LIN {X 0,Y 160.848,Z 396.644,A -85,B 0,C 180,E1 -25163.822,E2 -25163.822} C_VEL
LIN {X 0,Y 156.16,Z 389.326,A -85,B 0,C 180,E1 -25166.953,E2 -25166.953} C_VEL
LIN {X 0,Y 153.521,Z 385.51,A -85,B 0,C 180,E1 -25168.906,E2 -25168.906} C_VEL
LIN {X 0,Y 150.788,Z 381.597,A -85,B 0,C 180,E1 -25171.133,E2 -25171.133} C_VEL
LIN {X 0,Y 147.963,Z 377.724,A -85,B 0,C 180,E1 -25173.701,E2 -25173.701} C_VEL
LIN {X 0,Y 145.39,Z 374.72,A -85,B 0,C 180,E1 -25176.308,E2 -25176.308} C_VEL
LIN {X 0,Y 144.413,Z 372.921,A -85,B 0,C 180,E1 -25177.489,E2 -25177.489} C_VEL
LIN {X 0,Y 141.833,Z 370.706,A -85,B 0,C 180,E1 -25180.648,E2 -25180.648} C_VEL
LIN {X 0,Y 140.04,Z 367.443,A -85,B 0,C 180,E1 -25183.603,E2 -25183.603} C_VEL
LIN {X 0,Y 137.104,Z 365.186,A -85,B 0,C 180,E1 -25189.641,E2 -25189.641} C_VEL
LIN {X 0,Y 135.74,Z 362.249,A -85,B 0,C 180,E1 -25196.661,E2 -25196.661} C_VEL
LIN {X 0,Y 135.712,Z 361.677,A -85,B 0,C 180,E1 -25200,E2 -25200} C_VEL
LIN {X 0,Y 135.941,Z 362.758,A -85,B 0,C 180,E1 -25203.334,E2 -25203.334} C_VEL
LIN {X 0,Y 139.224,Z 367.011,A -85,B 0,C 180,E1 -25213.13,E2 -25213.13} C_VEL
LIN {X 0,Y 140.214,Z 367.722,A -85,B 0,C 180,E1 -25214.792,E2 -25214.792} C_VEL
LIN {X 0,Y 142.884,Z 372.468,A -85,B 0,C 180,E1 -25218.925,E2 -25218.925} C_VEL
LIN {X 0,Y 145.937,Z 377.229,A -85,B 0,C 180,E1 -25222.593,E2 -25222.593} C_VEL
LIN {X 0,Y 149.95,Z 384.374,A -85,B 0,C 180,E1 -25226.627,E2 -25226.627} C_VEL
LIN {X 0,Y 153.462,Z 391.115,A -85,B 0,C 180,E1 -25229.653,E2 -25229.653} C_VEL
LIN {X 0,Y 156.442,Z 397.18,A -85,B 0,C 180,E1 -25231.956,E2 -25231.956} C_VEL
LIN {X 0,Y 160.501,Z 406.172,A -85,B 0,C 180,E1 -25234.811,E2 -25234.811} C_VEL
LIN {X 0,Y 165.104,Z 417.859,A -85,B 0,C 180,E1 -25237.775,E2 -25237.775} C_VEL
LIN {X 0,Y 166.456,Z 421.823,A -85,B 0,C 180,E1 -25238.615,E2 -25238.615} C_VEL
LIN {X 0,Y 167.491,Z 450.285,A -85,B 0,C 180,E1 -25240.867,E2 -25240.867} C_VEL
LIN {X 0,Y 167.692,Z 465.573,A -85,B 0,C 180,E1 -25241.895,E2 -25241.895} C_VEL
LIN {X 0,Y 166.271,Z 479.287,A -85,B 0,C 180,E1 -25242.555,E2 -25242.555} C_VEL
LIN {X 0,Y 163.763,Z 492.886,A -85,B 0,C 180,E1 -25243.599,E2 -25243.599} C_VEL
LIN {X 0,Y 160.927,Z 503.892,A -85,B 0,C 180,E1 -25244.793,E2 -25244.793} C_VEL
LIN {X 0,Y 156.98,Z 515.737,A -85,B 0,C 180,E1 -25246.502,E2 -25246.502} C_VEL
LIN {X 0,Y 152.24,Z 527.599,A -85,B 0,C 180,E1 -25248.866,E2 -25248.866} C_VEL
LIN {X 0,Y 147.198,Z 538.138,A -85,B 0,C 180,E1 -25251.634,E2 -25251.634} C_VEL
LIN {X 0,Y 142.725,Z 546.719,A -85,B 0,C 180,E1 -25254.649,E2 -25254.649} C_VEL
LIN {X 0,Y 138.004,Z 555.138,A -85,B 0,C 180,E1 -25258.535,E2 -25258.535} C_VEL
LIN {X 0,Y 134.719,Z 560.938,A -85,B 0,C 180,E1 -25261.998,E2 -25261.998} C_VEL
LIN {X 0,Y 131.482,Z 566.642,A -85,B 0,C 180,E1 -25266.367,E2 -25266.367} C_VEL
LIN {X 0,Y 129.313,Z 571.196,A -85,B 0,C 180,E1 -25270.969,E2 -25270.969} C_VEL
LIN {X 0,Y 128.07,Z 574.695,A -85,B 0,C 180,E1 -25275.704,E2 -25275.704} C_VEL
LIN {X 0,Y 127.782,Z 577.781,A -85,B 0,C 180,E1 -25281.89,E2 -25281.89} C_VEL
LIN {X 0,Y 128.495,Z 579.127,A -85,B 0,C 180,E1 -25286.865,E2 -25286.865} C_VEL
LIN {X 0,Y 129.168,Z 579.454,A -85,B 0,C 180,E1 -25290,E2 -25290} C_VEL
LIN {X 0,Y 128.502,Z 579.112,A -85,B 0,C 180,E1 -25293.135,E2 -25293.135} C_VEL
LIN {X 0,Y 127.734,Z 577.185,A -85,B 0,C 180,E1 -25299.501,E2 -25299.501} C_VEL
LIN {X 0,Y 128.056,Z 574.636,A -85,B 0,C 180,E1 -25304.298,E2 -25304.298} C_VEL
LIN {X 0,Y 129.307,Z 571.111,A -85,B 0,C 180,E1 -25309.032,E2 -25309.032} C_VEL
LIN {X 0,Y 131.492,Z 566.532,A -85,B 0,C 180,E1 -25313.631,E2 -25313.631} C_VEL
LIN {X 0,Y 134.716,Z 560.8,A -85,B 0,C 180,E1 -25318.003,E2 -25318.003} C_VEL
LIN {X 0,Y 135.726,Z 559.01,A -85,B 0,C 180,E1 -25319.152,E2 -25319.152} C_VEL
LIN {X 0,Y 136.916,Z 555.737,A -85,B 0,C 180,E1 -25321.158,E2 -25321.158} C_VEL
LIN {X 0,Y 137.589,Z 549.959,A -85,B 0,C 180,E1 -25324.523,E2 -25324.523} C_VEL
LIN {X 0,Y 138.599,Z 543.677,A -85,B 0,C 180,E1 -25327.671,E2 -25327.671} C_VEL
LIN {X 0,Y 140.244,Z 539.563,A -85,B 0,C 180,E1 -25329.273,E2 -25329.273} C_VEL
LIN {X 0,Y 145.333,Z 529.702,A -85,B 0,C 180,E1 -25332.141,E2 -25332.141} C_VEL
LIN {X 0,Y 149.725,Z 520.009,A -85,B 0,C 180,E1 -25334.284,E2 -25334.284} C_VEL
LIN {X 0,Y 153.63,Z 509.578,A -85,B 0,C 180,E1 -25336.095,E2 -25336.095} C_VEL
LIN {X 0,Y 157.496,Z 497.125,A -85,B 0,C 180,E1 -25337.651,E2 -25337.651} C_VEL
LIN {X 0,Y 160.342,Z 484.282,A -85,B 0,C 180,E1 -25338.836,E2 -25338.836} C_VEL
LIN {X 0,Y 162.321,Z 470.908,A -85,B 0,C 180,E1 -25339.636,E2 -25339.636} C_VEL
LIN {X 0,Y 162.803,Z 463.571,A -85,B 0,C 180,E1 -25339.985,E2 -25339.985} C_VEL
LIN {X 0,Y 162.131,Z 433.785,A -85,B 0,C 180,E1 -25342.28,E2 -25342.28} C_VEL
LIN {X 0,Y 161.697,Z 423.97,A -85,B 0,C 180,E1 -25343.163,E2 -25343.163} C_VEL
LIN {X 0,Y 157.863,Z 413.397,A -85,B 0,C 180,E1 -25345.802,E2 -25345.802} C_VEL
LIN {X 0,Y 154.013,Z 404.075,A -85,B 0,C 180,E1 -25348.674,E2 -25348.674} C_VEL
LIN {X 0,Y 151.004,Z 397.589,A -85,B 0,C 180,E1 -25351.127,E2 -25351.127} C_VEL
LIN {X 0,Y 148.579,Z 392.638,A -85,B 0,C 180,E1 -25353.297,E2 -25353.297} C_VEL
LIN {X 0,Y 146.169,Z 387.847,A -85,B 0,C 180,E1 -25355.689,E2 -25355.689} C_VEL
LIN {X 0,Y 142.972,Z 381.909,A -85,B 0,C 180,E1 -25359.327,E2 -25359.327} C_VEL
LIN {X 0,Y 139.556,Z 376.178,A -85,B 0,C 180,E1 -25364.155,E2 -25364.155} C_VEL
LIN {X 0,Y 138.499,Z 374.182,A -85,B 0,C 180,E1 -25366.053,E2 -25366.053} C_VEL
LIN {X 0,Y 135.372,Z 370.964,A -85,B 0,C 180,E1 -25373.479,E2 -25373.479} C_VEL
LIN {X 0,Y 134.671,Z 368.946,A -85,B 0,C 180,E1 -25377.757,E2 -25377.757} C_VEL
LIN {X 0,Y 134.53,Z 368.503,A -85,B 0,C 180,E1 -25380,E2 -25380} C_VEL
LIN {X 0,Y 134.722,Z 369.26,A -85,B 0,C 180,E1 -25384.863,E2 -25384.863} C_VEL
LIN {X 0,Y 137.525,Z 373.69,A -85,B 0,C 180,E1 -25394.237,E2 -25394.237} C_VEL
LIN {X 0,Y 138.784,Z 374.55,A -85,B 0,C 180,E1 -25396.455,E2 -25396.455} C_VEL
LIN {X 0,Y 140.616,Z 377.811,A -85,B 0,C 180,E1 -25399.48,E2 -25399.48} C_VEL
LIN {X 0,Y 142.797,Z 379.938,A -85,B 0,C 180,E1 -25402.232,E2 -25402.232} C_VEL
LIN {X 0,Y 145.118,Z 383.369,A -85,B 0,C 180,E1 -25404.893,E2 -25404.893} C_VEL
LIN {X 0,Y 146.391,Z 384.854,A -85,B 0,C 180,E1 -25406.162,E2 -25406.162} C_VEL
LIN {X 0,Y 149.998,Z 390.076,A -85,B 0,C 180,E1 -25409.47,E2 -25409.47} C_VEL
LIN {X 0,Y 152.651,Z 394,A -85,B 0,C 180,E1 -25411.612,E2 -25411.612} C_VEL
LIN {X 0,Y 157.355,Z 401.577,A -85,B 0,C 180,E1 -25415.005,E2 -25415.005} C_VEL
LIN {X 0,Y 162.803,Z 411.309,A -85,B 0,C 180,E1 -25418.448,E2 -25418.448} C_VEL
LIN {X 0,Y 166.396,Z 418.787,A -85,B 0,C 180,E1 -25420.534,E2 -25420.534} C_VEL
LIN {X 0,Y 164.916,Z 443.762,A -85,B 0,C 180,E1 -25421.725,E2 -25421.725} C_VEL
LIN {X 0,Y 163.206,Z 456.855,A -85,B 0,C 180,E1 -25422.747,E2 -25422.747} C_VEL
LIN {X 0,Y 160.816,Z 468.889,A -85,B 0,C 180,E1 -25424.107,E2 -25424.107} C_VEL
LIN {X 0,Y 157.42,Z 481.198,A -85,B 0,C 180,E1 -25425.986,E2 -25425.986} C_VEL
LIN {X 0,Y 153.617,Z 491.66,A -85,B 0,C 180,E1 -25428.004,E2 -25428.004} C_VEL
LIN {X 0,Y 149.798,Z 500.707,A -85,B 0,C 180,E1 -25430.266,E2 -25430.266} C_VEL
LIN {X 0,Y 145.875,Z 509.102,A -85,B 0,C 180,E1 -25432.971,E2 -25432.971} C_VEL
LIN {X 0,Y 141.753,Z 516.834,A -85,B 0,C 180,E1 -25436.099,E2 -25436.099} C_VEL
LIN {X 0,Y 137.219,Z 524.484,A -85,B 0,C 180,E1 -25440.127,E2 -25440.127} C_VEL
LIN {X 0,Y 132.797,Z 531.281,A -85,B 0,C 180,E1 -25444.952,E2 -25444.952} C_VEL
LIN {X 0,Y 129.504,Z 535.886,A -85,B 0,C 180,E1 -25449.345,E2 -25449.345} C_VEL
LIN {X 0,Y 126.664,Z 539.432,A -85,B 0,C 180,E1 -25453.894,E2 -25453.894} C_VEL
LIN {X 0,Y 125.228,Z 541.253,A -85,B 0,C 180,E1 -25457.028,E2 -25457.028} C_VEL
LIN {X 0,Y 124.381,Z 542.581,A -85,B 0,C 180,E1 -25460.241,E2 -25460.241} C_VEL
LIN {X 0,Y 123.277,Z 544.125,A -85,B 0,C 180,E1 -25466.732,E2 -25466.732} C_VEL
LIN {X 0,Y 123.137,Z 544.345,A -85,B 0,C 180,E1 -25470,E2 -25470} C_VEL
LIN {X 0,Y 123.276,Z 544.154,A -85,B 0,C 180,E1 -25473.268,E2 -25473.268} C_VEL
LIN {X 0,Y 124.373,Z 542.648,A -85,B 0,C 180,E1 -25479.76,E2 -25479.76} C_VEL
LIN {X 0,Y 125.21,Z 541.351,A -85,B 0,C 180,E1 -25482.974,E2 -25482.974} C_VEL
LIN {X 0,Y 127.632,Z 538.503,A -85,B 0,C 180,E1 -25487.629,E2 -25487.629} C_VEL
LIN {X 0,Y 130.589,Z 534.667,A -85,B 0,C 180,E1 -25492.131,E2 -25492.131} C_VEL
LIN {X 0,Y 134.038,Z 529.576,A -85,B 0,C 180,E1 -25496.633,E2 -25496.633} C_VEL
LIN {X 0,Y 138.751,Z 522.322,A -85,B 0,C 180,E1 -25501.277,E2 -25501.277} C_VEL
LIN {X 0,Y 143.406,Z 514.284,A -85,B 0,C 180,E1 -25505.158,E2 -25505.158} C_VEL
LIN {X 0,Y 147.564,Z 506.049,A -85,B 0,C 180,E1 -25508.253,E2 -25508.253} C_VEL
LIN {X 0,Y 151.583,Z 496.997,A -85,B 0,C 180,E1 -25510.911,E2 -25510.911} C_VEL
LIN {X 0,Y 155.836,Z 486.44,A -85,B 0,C 180,E1 -25513.208,E2 -25513.208} C_VEL
LIN {X 0,Y 159.464,Z 474.891,A -85,B 0,C 180,E1 -25515.203,E2 -25515.203} C_VEL
LIN {X 0,Y 162.311,Z 463.568,A -85,B 0,C 180,E1 -25516.648,E2 -25516.648} C_VEL
LIN {X 0,Y 164.339,Z 450.783,A -85,B 0,C 180,E1 -25517.921,E2 -25517.921} C_VEL
LIN {X 0,Y 165.583,Z 437.335,A -85,B 0,C 180,E1 -25518.794,E2 -25518.794} C_VEL
LIN {X 0,Y 166.549,Z 418.84,A -85,B 0,C 180,E1 -25519.632,E2 -25519.632} C_VEL
LIN {X 0,Y 161.33,Z 408.377,A -85,B 0,C 180,E1 -25522.708,E2 -25522.708} C_VEL
LIN {X 0,Y 156.008,Z 399.158,A -85,B 0,C 180,E1 -25526.215,E2 -25526.215} C_VEL
LIN {X 0,Y 151.502,Z 392.096,A -85,B 0,C 180,E1 -25529.62,E2 -25529.62} C_VEL
LIN {X 0,Y 148.293,Z 387.477,A -85,B 0,C 180,E1 -25532.383,E2 -25532.383} C_VEL
LIN {X 0,Y 145.945,Z 384.127,A -85,B 0,C 180,E1 -25534.67,E2 -25534.67} C_VEL
LIN {X 0,Y 143.441,Z 380.953,A -85,B 0,C 180,E1 -25537.399,E2 -25537.399} C_VEL
LIN {X 0,Y 142.436,Z 379.406,A -85,B 0,C 180,E1 -25538.66,E2 -25538.66} C_VEL
LIN {X 0,Y 139.927,Z 376.762,A -85,B 0,C 180,E1 -25542.083,E2 -25542.083} C_VEL
LIN {X 0,Y 138.767,Z 374.319,A -85,B 0,C 180,E1 -25544.209,E2 -25544.209} C_VEL
LIN {X 0,Y 135.95,Z 371.966,A -85,B 0,C 180,E1 -25550.468,E2 -25550.468} C_VEL
LIN {X 0,Y 134.849,Z 369.244,A -85,B 0,C 180,E1 -25557.012,E2 -25557.012} C_VEL
LIN {X 0,Y 134.844,Z 368.749,A -85,B 0,C 180,E1 -25560,E2 -25560} C_VEL
LIN {X 0,Y 135.018,Z 369.778,A -85,B 0,C 180,E1 -25562.984,E2 -25562.984} C_VEL
LIN {X 0,Y 138.177,Z 373.995,A -85,B 0,C 180,E1 -25572.857,E2 -25572.857} C_VEL
LIN {X 0,Y 138.967,Z 374.761,A -85,B 0,C 180,E1 -25574.273,E2 -25574.273} C_VEL
LIN {X 0,Y 143.58,Z 382.67,A -85,B 0,C 180,E1 -25581.054,E2 -25581.054} C_VEL
LIN {X 0,Y 147.51,Z 390.237,A -85,B 0,C 180,E1 -25585.391,E2 -25585.391} C_VEL
LIN {X 0,Y 150.696,Z 396.745,A -85,B 0,C 180,E1 -25588.367,E2 -25588.367} C_VEL
LIN {X 0,Y 153.679,Z 403.119,A -85,B 0,C 180,E1 -25590.847,E2 -25590.847} C_VEL
LIN {X 0,Y 157.606,Z 412.501,A -85,B 0,C 180,E1 -25593.821,E2 -25593.821} C_VEL
LIN {X 0,Y 161.436,Z 422.806,A -85,B 0,C 180,E1 -25596.478,E2 -25596.478} C_VEL
LIN {X 0,Y 162.044,Z 424.806,A -85,B 0,C 180,E1 -25596.9,E2 -25596.9} C_VEL
LIN {X 0,Y 162.863,Z 454.654,A -85,B 0,C 180,E1 -25599.307,E2 -25599.307} C_VEL
LIN {X 0,Y 162.867,Z 466.599,A -85,B 0,C 180,E1 -25600.108,E2 -25600.108} C_VEL
LIN {X 0,Y 161.199,Z 480.534,A -85,B 0,C 180,E1 -25600.842,E2 -25600.842} C_VEL
LIN {X 0,Y 158.648,Z 493.207,A -85,B 0,C 180,E1 -25601.861,E2 -25601.861} C_VEL
LIN {X 0,Y 155.421,Z 504.815,A -85,B 0,C 180,E1 -25603.185,E2 -25603.185} C_VEL
LIN {X 0,Y 151.325,Z 516.187,A -85,B 0,C 180,E1 -25604.908,E2 -25604.908} C_VEL
LIN {X 0,Y 146.97,Z 526.615,A -85,B 0,C 180,E1 -25607.046,E2 -25607.046} C_VEL
LIN {X 0,Y 141.693,Z 537.151,A -85,B 0,C 180,E1 -25609.85,E2 -25609.85} C_VEL
LIN {X 0,Y 136.951,Z 545.726,A -85,B 0,C 180,E1 -25612.917,E2 -25612.917} C_VEL
LIN {X 0,Y 131.954,Z 554.144,A -85,B 0,C 180,E1 -25616.913,E2 -25616.913} C_VEL
LIN {X 0,Y 127.402,Z 561.729,A -85,B 0,C 180,E1 -25621.777,E2 -25621.777} C_VEL
LIN {X 0,Y 124.003,Z 567.302,A -85,B 0,C 180,E1 -25626.626,E2 -25626.626} C_VEL
LIN {X 0,Y 121.965,Z 571.498,A -85,B 0,C 180,E1 -25631.523,E2 -25631.523} C_VEL
LIN {X 0,Y 120.883,Z 574.668,A -85,B 0,C 180,E1 -25636.553,E2 -25636.553} C_VEL
LIN {X 0,Y 120.739,Z 576.9,A -85,B 0,C 180,E1 -25641.705,E2 -25641.705} C_VEL
LIN {X 0,Y 121.383,Z 578.136,A -85,B 0,C 180,E1 -25646.681,E2 -25646.681} C_VEL
LIN {X 0,Y 122.079,Z 578.468,A -85,B 0,C 180,E1 -25650,E2 -25650} C_VEL
LIN {X 0,Y 121.388,Z 578.12,A -85,B 0,C 180,E1 -25653.319,E2 -25653.319} C_VEL
LIN {X 0,Y 120.685,Z 576.189,A -85,B 0,C 180,E1 -25660.061,E2 -25660.061} C_VEL
LIN {X 0,Y 121.106,Z 573.635,A -85,B 0,C 180,E1 -25665.138,E2 -25665.138} C_VEL
LIN {X 0,Y 122.552,Z 570.113,A -85,B 0,C 180,E1 -25670.125,E2 -25670.125} C_VEL
LIN {X 0,Y 124.983,Z 565.537,A -85,B 0,C 180,E1 -25674.944,E2 -25674.944} C_VEL
LIN {X 0,Y 129.103,Z 558.739,A -85,B 0,C 180,E1 -25680.234,E2 -25680.234} C_VEL
LIN {X 0,Y 133.516,Z 551.342,A -85,B 0,C 180,E1 -25684.461,E2 -25684.461} C_VEL
LIN {X 0,Y 138.779,Z 542.234,A -85,B 0,C 180,E1 -25688.342,E2 -25688.342} C_VEL
LIN {X 0,Y 140.244,Z 539.563,A -85,B 0,C 180,E1 -25689.273,E2 -25689.273} C_VEL
LIN {X 0,Y 141.932,Z 535.289,A -85,B 0,C 180,E1 -25690.783,E2 -25690.783} C_VEL
LIN {X 0,Y 143.283,Z 527.963,A -85,B 0,C 180,E1 -25693.432,E2 -25693.432} C_VEL
LIN {X 0,Y 144.624,Z 520.254,A -85,B 0,C 180,E1 -25695.852,E2 -25695.852} C_VEL
LIN {X 0,Y 146.216,Z 515.282,A -85,B 0,C 180,E1 -25696.964,E2 -25696.964} C_VEL
LIN {X 0,Y 150.611,Z 503.291,A -85,B 0,C 180,E1 -25698.801,E2 -25698.801} C_VEL
LIN {X 0,Y 153.972,Z 491.422,A -85,B 0,C 180,E1 -25700.122,E2 -25700.122} C_VEL
LIN {X 0,Y 156.705,Z 477.922,A -85,B 0,C 180,E1 -25701.169,E2 -25701.169} C_VEL
LIN {X 0,Y 158.179,Z 465.114,A -85,B 0,C 180,E1 -25701.839,E2 -25701.839} C_VEL
LIN {X 0,Y 157.764,Z 435.791,A -85,B 0,C 180,E1 -25704.154,E2 -25704.154} C_VEL
LIN {X 0,Y 157.501,Z 427.116,A -85,B 0,C 180,E1 -25704.935,E2 -25704.935} C_VEL
LIN {X 0,Y 153.986,Z 417.044,A -85,B 0,C 180,E1 -25707.598,E2 -25707.598} C_VEL
LIN {X 0,Y 150.252,Z 407.681,A -85,B 0,C 180,E1 -25710.681,E2 -25710.681} C_VEL
LIN {X 0,Y 146.701,Z 399.622,A -85,B 0,C 180,E1 -25713.982,E2 -25713.982} C_VEL
LIN {X 0,Y 144.01,Z 393.968,A -85,B 0,C 180,E1 -25716.83,E2 -25716.83} C_VEL
LIN {X 0,Y 140.882,Z 387.867,A -85,B 0,C 180,E1 -25720.701,E2 -25720.701} C_VEL
LIN {X 0,Y 138.064,Z 382.758,A -85,B 0,C 180,E1 -25725.066,E2 -25725.066} C_VEL
LIN {X 0,Y 137.038,Z 380.911,A -85,B 0,C 180,E1 -25727.034,E2 -25727.034} C_VEL
LIN {X 0,Y 134.129,Z 377.356,A -85,B 0,C 180,E1 -25735.116,E2 -25735.116} C_VEL
LIN {X 0,Y 133.735,Z 375.85,A -85,B 0,C 180,E1 -25738.494,E2 -25738.494} C_VEL
LIN {X 0,Y 133.663,Z 375.564,A -85,B 0,C 180,E1 -25740,E2 -25740} C_VEL
LIN {X 0,Y 133.848,Z 376.404,A -85,B 0,C 180,E1 -25744.895,E2 -25744.895} C_VEL
LIN {X 0,Y 136.403,Z 380.62,A -85,B 0,C 180,E1 -25753.786,E2 -25753.786} C_VEL
LIN {X 0,Y 137.446,Z 381.457,A -85,B 0,C 180,E1 -25755.748,E2 -25755.748} C_VEL
LIN {X 0,Y 139.422,Z 384.832,A -85,B 0,C 180,E1 -25759.127,E2 -25759.127} C_VEL
LIN {X 0,Y 141.041,Z 386.461,A -85,B 0,C 180,E1 -25761.274,E2 -25761.274} C_VEL
LIN {X 0,Y 143.596,Z 390.188,A -85,B 0,C 180,E1 -25764.34,E2 -25764.34} C_VEL
LIN {X 0,Y 147.428,Z 395.805,A -85,B 0,C 180,E1 -25768.174,E2 -25768.174} C_VEL
LIN {X 0,Y 151.366,Z 401.899,A -85,B 0,C 180,E1 -25771.511,E2 -25771.511} C_VEL
LIN {X 0,Y 156.637,Z 411.198,A -85,B 0,C 180,E1 -25775.386,E2 -25775.386} C_VEL
LIN {X 0,Y 161.17,Z 420.199,A -85,B 0,C 180,E1 -25778.328,E2 -25778.328} C_VEL
LIN {X 0,Y 161.803,Z 421.629,A -85,B 0,C 180,E1 -25778.722,E2 -25778.722} C_VEL
LIN {X 0,Y 160.385,Z 444.105,A -85,B 0,C 180,E1 -25779.805,E2 -25779.805} C_VEL
LIN {X 0,Y 158.539,Z 457.708,A -85,B 0,C 180,E1 -25780.868,E2 -25780.868} C_VEL
LIN {X 0,Y 156.006,Z 469.873,A -85,B 0,C 180,E1 -25782.253,E2 -25782.253} C_VEL
LIN {X 0,Y 152.442,Z 482.184,A -85,B 0,C 180,E1 -25784.15,E2 -25784.15} C_VEL
LIN {X 0,Y 148.468,Z 492.642,A -85,B 0,C 180,E1 -25786.189,E2 -25786.189} C_VEL
LIN {X 0,Y 144.461,Z 501.689,A -85,B 0,C 180,E1 -25788.483,E2 -25788.483} C_VEL
LIN {X 0,Y 140.327,Z 510.083,A -85,B 0,C 180,E1 -25791.242,E2 -25791.242} C_VEL
LIN {X 0,Y 135.976,Z 517.814,A -85,B 0,C 180,E1 -25794.447,E2 -25794.447} C_VEL
LIN {X 0,Y 131.172,Z 525.464,A -85,B 0,C 180,E1 -25798.598,E2 -25798.598} C_VEL
LIN {X 0,Y 126.465,Z 532.261,A -85,B 0,C 180,E1 -25803.604,E2 -25803.604} C_VEL
LIN {X 0,Y 122.952,Z 536.865,A -85,B 0,C 180,E1 -25808.19,E2 -25808.19} C_VEL
LIN {X 0,Y 119.925,Z 540.411,A -85,B 0,C 180,E1 -25812.962,E2 -25812.962} C_VEL
LIN {X 0,Y 118.386,Z 542.232,A -85,B 0,C 180,E1 -25816.264,E2 -25816.264} C_VEL
LIN {X 0,Y 117.459,Z 543.56,A -85,B 0,C 180,E1 -25819.66,E2 -25819.66} C_VEL
LIN {X 0,Y 116.261,Z 545.103,A -85,B 0,C 180,E1 -25826.534,E2 -25826.534} C_VEL
LIN {X 0,Y 116.109,Z 545.323,A -85,B 0,C 180,E1 -25830,E2 -25830} C_VEL
LIN {X 0,Y 116.26,Z 545.131,A -85,B 0,C 180,E1 -25833.466,E2 -25833.466} C_VEL
LIN {X 0,Y 117.45,Z 543.626,A -85,B 0,C 180,E1 -25840.341,E2 -25840.341} C_VEL
LIN {X 0,Y 118.368,Z 542.329,A -85,B 0,C 180,E1 -25843.739,E2 -25843.739} C_VEL
LIN {X 0,Y 120.953,Z 539.481,A -85,B 0,C 180,E1 -25848.637,E2 -25848.637} C_VEL
LIN {X 0,Y 124.107,Z 535.644,A -85,B 0,C 180,E1 -25853.353,E2 -25853.353} C_VEL
LIN {X 0,Y 127.794,Z 530.552,A -85,B 0,C 180,E1 -25858.046,E2 -25858.046} C_VEL
LIN {X 0,Y 132.795,Z 523.298,A -85,B 0,C 180,E1 -25862.851,E2 -25862.851} C_VEL
LIN {X 0,Y 137.719,Z 515.259,A -85,B 0,C 180,E1 -25866.842,E2 -25866.842} C_VEL
LIN {X 0,Y 142.11,Z 507.024,A -85,B 0,C 180,E1 -25870.008,E2 -25870.008} C_VEL
LIN {X 0,Y 146.338,Z 497.972,A -85,B 0,C 180,E1 -25872.715,E2 -25872.715} C_VEL
LIN {X 0,Y 150.787,Z 487.415,A -85,B 0,C 180,E1 -25875.037,E2 -25875.037} C_VEL
LIN {X 0,Y 154.648,Z 475.706,A -85,B 0,C 180,E1 -25877.072,E2 -25877.072} C_VEL
LIN {X 0,Y 157.645,Z 464.191,A -85,B 0,C 180,E1 -25878.547,E2 -25878.547} C_VEL
LIN {X 0,Y 159.749,Z 451.455,A -85,B 0,C 180,E1 -25879.818,E2 -25879.818} C_VEL
LIN {X 0,Y 161.03,Z 438.419,A -85,B 0,C 180,E1 -25880.67,E2 -25880.67} C_VEL
LIN {X 0,Y 161.949,Z 421.662,A -85,B 0,C 180,E1 -25881.455,E2 -25881.455} C_VEL
LIN {X 0,Y 157.147,Z 411.982,A -85,B 0,C 180,E1 -25884.55,E2 -25884.55} C_VEL
LIN {X 0,Y 152.314,Z 403.442,A -85,B 0,C 180,E1 -25888.049,E2 -25888.049} C_VEL
LIN {X 0,Y 148.448,Z 397.272,A -85,B 0,C 180,E1 -25891.251,E2 -25891.251} C_VEL
LIN {X 0,Y 146.093,Z 393.664,A -85,B 0,C 180,E1 -25893.458,E2 -25893.458} C_VEL
LIN {X 0,Y 143.952,Z 390.483,A -85,B 0,C 180,E1 -25895.688,E2 -25895.688} C_VEL
LIN {X 0,Y 141.48,Z 387.094,A -85,B 0,C 180,E1 -25898.605,E2 -25898.605} C_VEL
LIN {X 0,Y 140.583,Z 385.89,A -85,B 0,C 180,E1 -25899.792,E2 -25899.792} C_VEL
LIN {X 0,Y 138.115,Z 382.793,A -85,B 0,C 180,E1 -25903.558,E2 -25903.558} C_VEL
LIN {X 0,Y 137.312,Z 381.111,A -85,B 0,C 180,E1 -25905.172,E2 -25905.172} C_VEL
LIN {X 0,Y 134.649,Z 378.388,A -85,B 0,C 180,E1 -25912.03,E2 -25912.03} C_VEL
LIN {X 0,Y 133.95,Z 376.155,A -85,B 0,C 180,E1 -25917.745,E2 -25917.745} C_VEL
LIN {X 0,Y 133.975,Z 375.823,A -85,B 0,C 180,E1 -25920,E2 -25920} C_VEL
LIN {X 0,Y 134.243,Z 377.324,A -85,B 0,C 180,E1 -25923.846,E2 -25923.846} C_VEL
LIN {X 0,Y 137.037,Z 380.928,A -85,B 0,C 180,E1 -25932.401,E2 -25932.401} C_VEL
LIN {X 0,Y 137.596,Z 381.543,A -85,B 0,C 180,E1 -25933.476,E2 -25933.476} C_VEL
LIN {X 0,Y 141.593,Z 388.885,A -85,B 0,C 180,E1 -25939.858,E2 -25939.858} C_VEL
LIN {X 0,Y 145.11,Z 396.031,A -85,B 0,C 180,E1 -25944.08,E2 -25944.08} C_VEL
LIN {X 0,Y 148.079,Z 402.456,A -85,B 0,C 180,E1 -25947.093,E2 -25947.093} C_VEL
LIN {X 0,Y 150.761,Z 408.567,A -85,B 0,C 180,E1 -25949.517,E2 -25949.517} C_VEL
LIN {X 0,Y 154.897,Z 419.086,A -85,B 0,C 180,E1 -25952.891,E2 -25952.891} C_VEL
LIN {X 0,Y 157.708,Z 427.283,A -85,B 0,C 180,E1 -25955.012,E2 -25955.012} C_VEL
LIN {X 0,Y 158.284,Z 452.976,A -85,B 0,C 180,E1 -25957.187,E2 -25957.187} C_VEL
LIN {X 0,Y 158.332,Z 465.877,A -85,B 0,C 180,E1 -25958.14,E2 -25958.14} C_VEL
LIN {X 0,Y 156.635,Z 479.443,A -85,B 0,C 180,E1 -25958.856,E2 -25958.856} C_VEL
LIN {X 0,Y 154.057,Z 491.955,A -85,B 0,C 180,E1 -25959.864,E2 -25959.864} C_VEL
LIN {X 0,Y 150.637,Z 503.83,A -85,B 0,C 180,E1 -25961.21,E2 -25961.21} C_VEL
LIN {X 0,Y 146.398,Z 515.203,A -85,B 0,C 180,E1 -25962.939,E2 -25962.939} C_VEL
LIN {X 0,Y 141.284,Z 526.813,A -85,B 0,C 180,E1 -25965.362,E2 -25965.362} C_VEL
LIN {X 0,Y 136.343,Z 536.166,A -85,B 0,C 180,E1 -25967.926,E2 -25967.926} C_VEL
LIN {X 0,Y 131.325,Z 544.735,A -85,B 0,C 180,E1 -25971.038,E2 -25971.038} C_VEL
LIN {X 0,Y 126.034,Z 553.153,A -85,B 0,C 180,E1 -25975.141,E2 -25975.141} C_VEL
LIN {X 0,Y 121.561,Z 560.069,A -85,B 0,C 180,E1 -25979.678,E2 -25979.678} C_VEL
LIN {X 0,Y 117.47,Z 566.307,A -85,B 0,C 180,E1 -25985.242,E2 -25985.242} C_VEL
LIN {X 0,Y 115.186,Z 570.501,A -85,B 0,C 180,E1 -25990.393,E2 -25990.393} C_VEL
LIN {X 0,Y 113.901,Z 573.668,A -85,B 0,C 180,E1 -25995.711,E2 -25995.711} C_VEL
LIN {X 0,Y 113.75,Z 576.381,A -85,B 0,C 180,E1 -26002.902,E2 -26002.902} C_VEL
LIN {X 0,Y 114.256,Z 577.142,A -85,B 0,C 180,E1 -26006.473,E2 -26006.473} C_VEL
LIN {X 0,Y 114.986,Z 577.481,A -85,B 0,C 180,E1 -26010,E2 -26010} C_VEL
LIN {X 0,Y 114.26,Z 577.127,A -85,B 0,C 180,E1 -26013.526,E2 -26013.526} C_VEL
LIN {X 0,Y 113.624,Z 575.19,A -85,B 0,C 180,E1 -26020.694,E2 -26020.694} C_VEL
LIN {X 0,Y 114.208,Z 572.638,A -85,B 0,C 180,E1 -26026.076,E2 -26026.076} C_VEL
LIN {X 0,Y 115.848,Z 569.114,A -85,B 0,C 180,E1 -26031.345,E2 -26031.345} C_VEL
LIN {X 0,Y 118.552,Z 564.543,A -85,B 0,C 180,E1 -26036.398,E2 -26036.398} C_VEL
LIN {X 0,Y 122.281,Z 558.808,A -85,B 0,C 180,E1 -26041.148,E2 -26041.148} C_VEL
LIN {X 0,Y 126.824,Z 551.705,A -85,B 0,C 180,E1 -26045.581,E2 -26045.581} C_VEL
LIN {X 0,Y 132.271,Z 542.891,A -85,B 0,C 180,E1 -26049.612,E2 -26049.612} C_VEL
LIN {X 0,Y 137.428,Z 533.921,A -85,B 0,C 180,E1 -26052.655,E2 -26052.655} C_VEL
LIN {X 0,Y 142.445,Z 524.105,A -85,B 0,C 180,E1 -26055.172,E2 -26055.172} C_VEL
LIN {X 0,Y 146.216,Z 515.282,A -85,B 0,C 180,E1 -26056.964,E2 -26056.964} C_VEL
LIN {X 0,Y 147.704,Z 510.207,A -85,B 0,C 180,E1 -26058.001,E2 -26058.001} C_VEL
LIN {X 0,Y 148.584,Z 501.748,A -85,B 0,C 180,E1 -26059.993,E2 -26059.993} C_VEL
LIN {X 0,Y 149.261,Z 492.996,A -85,B 0,C 180,E1 -26061.776,E2 -26061.776} C_VEL
LIN {X 0,Y 150.229,Z 487.462,A -85,B 0,C 180,E1 -26062.481,E2 -26062.481} C_VEL
LIN {X 0,Y 152.716,Z 474.548,A -85,B 0,C 180,E1 -26063.408,E2 -26063.408} C_VEL
LIN {X 0,Y 153.739,Z 465.227,A -85,B 0,C 180,E1 -26063.893,E2 -26063.893} C_VEL
LIN {X 0,Y 153.516,Z 432.78,A -85,B 0,C 180,E1 -26066.569,E2 -26066.569} C_VEL
LIN {X 0,Y 153.362,Z 429.815,A -85,B 0,C 180,E1 -26066.894,E2 -26066.894} C_VEL
LIN {X 0,Y 149.536,Z 418.574,A -85,B 0,C 180,E1 -26070.139,E2 -26070.139} C_VEL
LIN {X 0,Y 145.846,Z 409.204,A -85,B 0,C 180,E1 -26073.626,E2 -26073.626} C_VEL
LIN {X 0,Y 143.101,Z 402.828,A -85,B 0,C 180,E1 -26076.578,E2 -26076.578} C_VEL
LIN {X 0,Y 141.421,Z 399.173,A -85,B 0,C 180,E1 -26078.595,E2 -26078.595} C_VEL
LIN {X 0,Y 138.973,Z 393.977,A -85,B 0,C 180,E1 -26081.977,E2 -26081.977} C_VEL
LIN {X 0,Y 136.318,Z 388.733,A -85,B 0,C 180,E1 -26086.585,E2 -26086.585} C_VEL
LIN {X 0,Y 135.798,Z 387.799,A -85,B 0,C 180,E1 -26087.674,E2 -26087.674} C_VEL
LIN {X 0,Y 133.076,Z 383.96,A -85,B 0,C 180,E1 -26096.215,E2 -26096.215} C_VEL
LIN {X 0,Y 132.819,Z 382.777,A -85,B 0,C 180,E1 -26099.242,E2 -26099.242} C_VEL
LIN {X 0,Y 132.817,Z 382.969,A -85,B 0,C 180,E1 -26103.033,E2 -26103.033} C_VEL
LIN {X 0,Y 133.194,Z 384.412,A -85,B 0,C 180,E1 -26106.612,E2 -26106.612} C_VEL
LIN {X 0,Y 135.555,Z 387.731,A -85,B 0,C 180,E1 -26113.874,E2 -26113.874} C_VEL
LIN {X 0,Y 136.103,Z 388.271,A -85,B 0,C 180,E1 -26114.963,E2 -26114.963} C_VEL
LIN {X 0,Y 138.207,Z 391.802,A -85,B 0,C 180,E1 -26118.724,E2 -26118.724} C_VEL
LIN {X 0,Y 139.51,Z 393.286,A -85,B 0,C 180,E1 -26120.552,E2 -26120.552} C_VEL
LIN {X 0,Y 142.607,Z 397.962,A -85,B 0,C 180,E1 -26124.387,E2 -26124.387} C_VEL
LIN {X 0,Y 145.494,Z 402.471,A -85,B 0,C 180,E1 -26127.386,E2 -26127.386} C_VEL
LIN {X 0,Y 148.757,Z 407.719,A -85,B 0,C 180,E1 -26130.327,E2 -26130.327} C_VEL
LIN {X 0,Y 153.501,Z 416.527,A -85,B 0,C 180,E1 -26134.086,E2 -26134.086} C_VEL
LIN {X 0,Y 157.394,Z 424.586,A -85,B 0,C 180,E1 -26136.822,E2 -26136.822} C_VEL
LIN {X 0,Y 155.964,Z 445.163,A -85,B 0,C 180,E1 -26137.822,E2 -26137.822} C_VEL
LIN {X 0,Y 154.001,Z 458.836,A -85,B 0,C 180,E1 -26138.9,E2 -26138.9} C_VEL
LIN {X 0,Y 151.37,Z 470.858,A -85,B 0,C 180,E1 -26140.283,E2 -26140.283} C_VEL
LIN {X 0,Y 147.964,Z 482.19,A -85,B 0,C 180,E1 -26142.016,E2 -26142.016} C_VEL
LIN {X 0,Y 144.011,Z 492.354,A -85,B 0,C 180,E1 -26143.961,E2 -26143.961} C_VEL
LIN {X 0,Y 139.752,Z 501.627,A -85,B 0,C 180,E1 -26146.254,E2 -26146.254} C_VEL
LIN {X 0,Y 134.917,Z 511.064,A -85,B 0,C 180,E1 -26149.373,E2 -26149.373} C_VEL
LIN {X 0,Y 130.322,Z 518.794,A -85,B 0,C 180,E1 -26152.65,E2 -26152.65} C_VEL
LIN {X 0,Y 125.227,Z 526.444,A -85,B 0,C 180,E1 -26156.922,E2 -26156.922} C_VEL
LIN {X 0,Y 120.211,Z 533.24,A -85,B 0,C 180,E1 -26162.115,E2 -26162.115} C_VEL
LIN {X 0,Y 116.457,Z 537.844,A -85,B 0,C 180,E1 -26166.905,E2 -26166.905} C_VEL
LIN {X 0,Y 113.221,Z 541.39,A -85,B 0,C 180,E1 -26171.919,E2 -26171.919} C_VEL
LIN {X 0,Y 111.568,Z 543.212,A -85,B 0,C 180,E1 -26175.406,E2 -26175.406} C_VEL
LIN {X 0,Y 110.55,Z 544.539,A -85,B 0,C 180,E1 -26179.006,E2 -26179.006} C_VEL
LIN {X 0,Y 109.246,Z 546.081,A -85,B 0,C 180,E1 -26186.312,E2 -26186.312} C_VEL
LIN {X 0,Y 109.081,Z 546.301,A -85,B 0,C 180,E1 -26190,E2 -26190} C_VEL
LIN {X 0,Y 109.246,Z 546.109,A -85,B 0,C 180,E1 -26193.688,E2 -26193.688} C_VEL
LIN {X 0,Y 110.542,Z 544.604,A -85,B 0,C 180,E1 -26200.995,E2 -26200.995} C_VEL
LIN {X 0,Y 111.549,Z 543.307,A -85,B 0,C 180,E1 -26204.596,E2 -26204.596} C_VEL
LIN {X 0,Y 114.316,Z 540.458,A -85,B 0,C 180,E1 -26209.763,E2 -26209.763} C_VEL
LIN {X 0,Y 117.687,Z 536.621,A -85,B 0,C 180,E1 -26214.709,E2 -26214.709} C_VEL
LIN {X 0,Y 121.637,Z 531.528,A -85,B 0,C 180,E1 -26219.602,E2 -26219.602} C_VEL
LIN {X 0,Y 126.948,Z 524.274,A -85,B 0,C 180,E1 -26224.572,E2 -26224.572} C_VEL
LIN {X 0,Y 132.161,Z 516.235,A -85,B 0,C 180,E1 -26228.67,E2 -26228.67} C_VEL
LIN {X 0,Y 136.8,Z 508,A -85,B 0,C 180,E1 -26231.902,E2 -26231.902} C_VEL
LIN {X 0,Y 141.251,Z 498.947,A -85,B 0,C 180,E1 -26234.651,E2 -26234.651} C_VEL
LIN {X 0,Y 145.907,Z 488.387,A -85,B 0,C 180,E1 -26236.99,E2 -26236.99} C_VEL
LIN {X 0,Y 149.95,Z 476.678,A -85,B 0,C 180,E1 -26239.039,E2 -26239.039} C_VEL
LIN {X 0,Y 153.085,Z 465.161,A -85,B 0,C 180,E1 -26240.518,E2 -26240.518} C_VEL
LIN {X 0,Y 155.288,Z 452.467,A -85,B 0,C 180,E1 -26241.802,E2 -26241.802} C_VEL
LIN {X 0,Y 156.723,Z 438.692,A -85,B 0,C 180,E1 -26242.693,E2 -26242.693} C_VEL
LIN {X 0,Y 157.53,Z 424.652,A -85,B 0,C 180,E1 -26243.366,E2 -26243.366} C_VEL
LIN {X 0,Y 153.043,Z 415.396,A -85,B 0,C 180,E1 -26246.56,E2 -26246.56} C_VEL
LIN {X 0,Y 148.454,Z 407.109,A -85,B 0,C 180,E1 -26250.263,E2 -26250.263} C_VEL
LIN {X 0,Y 144.221,Z 400.165,A -85,B 0,C 180,E1 -26254.289,E2 -26254.289} C_VEL
LIN {X 0,Y 141.901,Z 396.745,A -85,B 0,C 180,E1 -26256.851,E2 -26256.851} C_VEL
LIN {X 0,Y 139.201,Z 392.703,A -85,B 0,C 180,E1 -26260.384,E2 -26260.384} C_VEL
LIN {X 0,Y 136.749,Z 389.52,A -85,B 0,C 180,E1 -26264.347,E2 -26264.347} C_VEL
LIN {X 0,Y 136.083,Z 387.982,A -85,B 0,C 180,E1 -26265.799,E2 -26265.799} C_VEL
LIN {X 0,Y 133.67,Z 385.365,A -85,B 0,C 180,E1 -26272.447,E2 -26272.447} C_VEL
LIN {X 0,Y 133.08,Z 383.248,A -85,B 0,C 180,E1 -26277.73,E2 -26277.73} C_VEL
LIN {X 0,Y 133.12,Z 383.02,A -85,B 0,C 180,E1 -26280.567,E2 -26280.567} C_VEL
LIN {X 0,Y 135.906,Z 387.859,A -85,B 0,C 180,E1 -26291.938,E2 -26291.938} C_VEL
LIN {X 0,Y 136.501,Z 388.897,A -85,B 0,C 180,E1 -26293.207,E2 -26293.207} C_VEL
LIN {X 0,Y 139.724,Z 395.176,A -85,B 0,C 180,E1 -26298.703,E2 -26298.703} C_VEL
LIN {X 0,Y 142.824,Z 401.914,A -85,B 0,C 180,E1 -26302.769,E2 -26302.769} C_VEL
LIN {X 0,Y 145.687,Z 408.59,A -85,B 0,C 180,E1 -26305.935,E2 -26305.935} C_VEL
LIN {X 0,Y 148.47,Z 415.37,A -85,B 0,C 180,E1 -26308.638,E2 -26308.638} C_VEL
LIN {X 0,Y 152.273,Z 426.062,A -85,B 0,C 180,E1 -26311.987,E2 -26311.987} C_VEL
LIN {X 0,Y 153.627,Z 430.224,A -85,B 0,C 180,E1 -26313.1,E2 -26313.1} C_VEL
LIN {X 0,Y 153.965,Z 458.025,A -85,B 0,C 180,E1 -26315.482,E2 -26315.482} C_VEL
LIN {X 0,Y 153.77,Z 467.829,A -85,B 0,C 180,E1 -26316.188,E2 -26316.188} C_VEL
LIN {X 0,Y 151.841,Z 481.014,A -85,B 0,C 180,E1 -26316.949,E2 -26316.949} C_VEL
LIN {X 0,Y 148.813,Z 493.757,A -85,B 0,C 180,E1 -26318.043,E2 -26318.043} C_VEL
LIN {X 0,Y 144.803,Z 506.4,A -85,B 0,C 180,E1 -26319.603,E2 -26319.603} C_VEL
LIN {X 0,Y 139.802,Z 518.39,A -85,B 0,C 180,E1 -26321.602,E2 -26321.602} C_VEL
LIN {X 0,Y 135.139,Z 528.042,A -85,B 0,C 180,E1 -26323.816,E2 -26323.816} C_VEL
LIN {X 0,Y 128.96,Z 538.795,A -85,B 0,C 180,E1 -26327.062,E2 -26327.062} C_VEL
LIN {X 0,Y 123.923,Z 546.774,A -85,B 0,C 180,E1 -26330.357,E2 -26330.357} C_VEL
LIN {X 0,Y 118.544,Z 554.608,A -85,B 0,C 180,E1 -26334.688,E2 -26334.688} C_VEL
LIN {X 0,Y 113.442,Z 561.911,A -85,B 0,C 180,E1 -26340.29,E2 -26340.29} C_VEL
LIN {X 0,Y 110.039,Z 566.818,A -85,B 0,C 180,E1 -26345.472,E2 -26345.472} C_VEL
LIN {X 0,Y 107.837,Z 570.653,A -85,B 0,C 180,E1 -26350.982,E2 -26350.982} C_VEL
LIN {X 0,Y 106.971,Z 572.672,A -85,B 0,C 180,E1 -26354.764,E2 -26354.764} C_VEL
LIN {X 0,Y 106.669,Z 575.388,A -85,B 0,C 180,E1 -26362.428,E2 -26362.428} C_VEL
LIN {X 0,Y 107.136,Z 576.15,A -85,B 0,C 180,E1 -26366.239,E2 -26366.239} C_VEL
LIN {X 0,Y 107.886,Z 576.493,A -85,B 0,C 180,E1 -26370,E2 -26370} C_VEL
LIN {X 0,Y 107.14,Z 576.134,A -85,B 0,C 180,E1 -26373.761,E2 -26373.761} C_VEL
LIN {X 0,Y 106.621,Z 575.101,A -85,B 0,C 180,E1 -26378.608,E2 -26378.608} C_VEL
LIN {X 0,Y 106.96,Z 572.616,A -85,B 0,C 180,E1 -26385.238,E2 -26385.238} C_VEL
LIN {X 0,Y 108.461,Z 569.427,A -85,B 0,C 180,E1 -26390.878,E2 -26390.878} C_VEL
LIN {X 0,Y 111.028,Z 565.209,A -85,B 0,C 180,E1 -26396.301,E2 -26396.301} C_VEL
LIN {X 0,Y 115.404,Z 558.956,A -85,B 0,C 180,E1 -26402.096,E2 -26402.096} C_VEL
LIN {X 0,Y 120.201,Z 551.972,A -85,B 0,C 180,E1 -26406.819,E2 -26406.819} C_VEL
LIN {X 0,Y 125.863,Z 543.524,A -85,B 0,C 180,E1 -26411.002,E2 -26411.002} C_VEL
LIN {X 0,Y 131.164,Z 534.899,A -85,B 0,C 180,E1 -26414.151,E2 -26414.151} C_VEL
LIN {X 0,Y 136.934,Z 524.296,A -85,B 0,C 180,E1 -26417,E2 -26417} C_VEL
LIN {X 0,Y 141.668,Z 513.793,A -85,B 0,C 180,E1 -26419.159,E2 -26419.159} C_VEL
LIN {X 0,Y 145.957,Z 502.523,A -85,B 0,C 180,E1 -26420.866,E2 -26420.866} C_VEL
LIN {X 0,Y 149.598,Z 490.039,A -85,B 0,C 180,E1 -26422.252,E2 -26422.252} C_VEL
LIN {X 0,Y 150.229,Z 487.462,A -85,B 0,C 180,E1 -26422.481,E2 -26422.481} C_VEL
LIN {X 0,Y 151.109,Z 481.848,A -85,B 0,C 180,E1 -26423.104,E2 -26423.104} C_VEL
LIN {X 0,Y 151.151,Z 476.312,A -85,B 0,C 180,E1 -26423.93,E2 -26423.93} C_VEL
LIN {X 0,Y 149.776,Z 461.546,A -85,B 0,C 180,E1 -26426.267,E2 -26426.267} C_VEL
LIN {X 0,Y 149.587,Z 457.692,A -85,B 0,C 180,E1 -26426.692,E2 -26426.692} C_VEL
LIN {X 0,Y 149.5,Z 433.017,A -85,B 0,C 180,E1 -26428.861,E2 -26428.861} C_VEL
LIN {X 0,Y 146.222,Z 422.872,A -85,B 0,C 180,E1 -26431.958,E2 -26431.958} C_VEL
LIN {X 0,Y 143.185,Z 414.567,A -85,B 0,C 180,E1 -26435.148,E2 -26435.148} C_VEL
LIN {X 0,Y 140.067,Z 406.647,A -85,B 0,C 180,E1 -26438.957,E2 -26438.957} C_VEL
LIN {X 0,Y 137.05,Z 399.913,A -85,B 0,C 180,E1 -26443.426,E2 -26443.426} C_VEL
LIN {X 0,Y 134.745,Z 394.904,A -85,B 0,C 180,E1 -26447.958,E2 -26447.958} C_VEL
LIN {X 0,Y 131.951,Z 389.85,A -85,B 0,C 180,E1 -26459.237,E2 -26459.237} C_VEL
LIN {X 0,Y 131.949,Z 390.045,A -85,B 0,C 180,E1 -26463.053,E2 -26463.053} C_VEL
LIN {X 0,Y 134.352,Z 394.609,A -85,B 0,C 180,E1 -26473.23,E2 -26473.23} C_VEL
LIN {X 0,Y 134.882,Z 395.27,A -85,B 0,C 180,E1 -26474.378,E2 -26474.378} C_VEL
LIN {X 0,Y 136.999,Z 398.771,A -85,B 0,C 180,E1 -26478.313,E2 -26478.313} C_VEL
LIN {X 0,Y 137.956,Z 400.051,A -85,B 0,C 180,E1 -26479.75,E2 -26479.75} C_VEL
LIN {X 0,Y 140.757,Z 404.462,A -85,B 0,C 180,E1 -26483.446,E2 -26483.446} C_VEL
LIN {X 0,Y 143.705,Z 409.278,A -85,B 0,C 180,E1 -26486.689,E2 -26486.689} C_VEL
LIN {X 0,Y 147.548,Z 416.079,A -85,B 0,C 180,E1 -26490.305,E2 -26490.305} C_VEL
LIN {X 0,Y 151.962,Z 424.943,A -85,B 0,C 180,E1 -26493.909,E2 -26493.909} C_VEL
LIN {X 0,Y 153.12,Z 427.513,A -85,B 0,C 180,E1 -26494.786,E2 -26494.786} C_VEL
LIN {X 0,Y 151.665,Z 446.93,A -85,B 0,C 180,E1 -26495.775,E2 -26495.775} C_VEL
LIN {X 0,Y 149.762,Z 459.446,A -85,B 0,C 180,E1 -26496.773,E2 -26496.773} C_VEL
LIN {X 0,Y 146.954,Z 471.743,A -85,B 0,C 180,E1 -26498.18,E2 -26498.18} C_VEL
LIN {X 0,Y 143.423,Z 482.98,A -85,B 0,C 180,E1 -26499.893,E2 -26499.893} C_VEL
LIN {X 0,Y 139.224,Z 493.336,A -85,B 0,C 180,E1 -26501.879,E2 -26501.879} C_VEL
LIN {X 0,Y 134.76,Z 502.609,A -85,B 0,C 180,E1 -26504.187,E2 -26504.187} C_VEL
LIN {X 0,Y 129.663,Z 512.045,A -85,B 0,C 180,E1 -26507.35,E2 -26507.35} C_VEL
LIN {X 0,Y 124.807,Z 519.775,A -85,B 0,C 180,E1 -26510.692,E2 -26510.692} C_VEL
LIN {X 0,Y 119.399,Z 527.423,A -85,B 0,C 180,E1 -26515.081,E2 -26515.081} C_VEL
LIN {X 0,Y 114.046,Z 534.22,A -85,B 0,C 180,E1 -26520.463,E2 -26520.463} C_VEL
LIN {X 0,Y 110.026,Z 538.823,A -85,B 0,C 180,E1 -26525.469,E2 -26525.469} C_VEL
LIN {X 0,Y 106.559,Z 542.37,A -85,B 0,C 180,E1 -26530.746,E2 -26530.746} C_VEL
LIN {X 0,Y 104.778,Z 544.191,A -85,B 0,C 180,E1 -26534.437,E2 -26534.437} C_VEL
LIN {X 0,Y 103.658,Z 545.517,A -85,B 0,C 180,E1 -26538.264,E2 -26538.264} C_VEL
LIN {X 0,Y 102.234,Z 547.059,A -85,B 0,C 180,E1 -26546.058,E2 -26546.058} C_VEL
LIN {X 0,Y 102.053,Z 547.279,A -85,B 0,C 180,E1 -26550,E2 -26550} C_VEL
LIN {X 0,Y 102.233,Z 547.087,A -85,B 0,C 180,E1 -26553.942,E2 -26553.942} C_VEL
LIN {X 0,Y 103.65,Z 545.581,A -85,B 0,C 180,E1 -26561.737,E2 -26561.737} C_VEL
LIN {X 0,Y 104.759,Z 544.285,A -85,B 0,C 180,E1 -26565.566,E2 -26565.566} C_VEL
LIN {X 0,Y 107.728,Z 541.435,A -85,B 0,C 180,E1 -26571.027,E2 -26571.027} C_VEL
LIN {X 0,Y 111.341,Z 537.597,A -85,B 0,C 180,E1 -26576.221,E2 -26576.221} C_VEL
LIN {X 0,Y 115.578,Z 532.505,A -85,B 0,C 180,E1 -26581.324,E2 -26581.324} C_VEL
LIN {X 0,Y 121.227,Z 525.25,A -85,B 0,C 180,E1 -26586.457,E2 -26586.457} C_VEL
LIN {X 0,Y 126.749,Z 517.211,A -85,B 0,C 180,E1 -26590.655,E2 -26590.655} C_VEL
LIN {X 0,Y 131.651,Z 508.975,A -85,B 0,C 180,E1 -26593.946,E2 -26593.946} C_VEL
LIN {X 0,Y 136.345,Z 499.921,A -85,B 0,C 180,E1 -26596.725,E2 -26596.725} C_VEL
LIN {X 0,Y 141.208,Z 489.36,A -85,B 0,C 180,E1 -26599.075,E2 -26599.075} C_VEL
LIN {X 0,Y 145.381,Z 477.807,A -85,B 0,C 180,E1 -26601.11,E2 -26601.11} C_VEL
LIN {X 0,Y 148.638,Z 466.478,A -85,B 0,C 180,E1 -26602.565,E2 -26602.565} C_VEL
LIN {X 0,Y 150.931,Z 454.15,A -85,B 0,C 180,E1 -26603.844,E2 -26603.844} C_VEL
LIN {X 0,Y 152.488,Z 440.902,A -85,B 0,C 180,E1 -26604.714,E2 -26604.714} C_VEL
LIN {X 0,Y 153.232,Z 427.479,A -85,B 0,C 180,E1 -26605.434,E2 -26605.434} C_VEL
LIN {X 0,Y 148.943,Z 418.595,A -85,B 0,C 180,E1 -26608.827,E2 -26608.827} C_VEL
LIN {X 0,Y 145.072,Z 411.419,A -85,B 0,C 180,E1 -26612.329,E2 -26612.329} C_VEL
LIN {X 0,Y 141.706,Z 405.773,A -85,B 0,C 180,E1 -26615.878,E2 -26615.878} C_VEL
LIN {X 0,Y 139.77,Z 402.754,A -85,B 0,C 180,E1 -26618.233,E2 -26618.233} C_VEL
LIN {X 0,Y 137.546,Z 399.239,A -85,B 0,C 180,E1 -26621.408,E2 -26621.408} C_VEL
LIN {X 0,Y 135.244,Z 395.89,A -85,B 0,C 180,E1 -26625.517,E2 -26625.517} C_VEL
LIN {X 0,Y 134.692,Z 394.772,A -85,B 0,C 180,E1 -26626.804,E2 -26626.804} C_VEL
LIN {X 0,Y 132.204,Z 390.242,A -85,B 0,C 180,E1 -26638.115,E2 -26638.115} C_VEL
LIN {X 0,Y 132.243,Z 390.076,A -85,B 0,C 180,E1 -26640.38,E2 -26640.38} C_VEL
LIN {X 0,Y 134.697,Z 394.726,A -85,B 0,C 180,E1 -26651.283,E2 -26651.283} C_VEL
LIN {X 0,Y 135.809,Z 396.979,A -85,B 0,C 180,E1 -26653.752,E2 -26653.752} C_VEL
LIN {X 0,Y 137.968,Z 401.598,A -85,B 0,C 180,E1 -26657.605,E2 -26657.605} C_VEL
LIN {X 0,Y 140.67,Z 407.981,A -85,B 0,C 180,E1 -26661.494,E2 -26661.494} C_VEL
LIN {X 0,Y 143.35,Z 414.649,A -85,B 0,C 180,E1 -26664.725,E2 -26664.725} C_VEL
LIN {X 0,Y 146.447,Z 423.07,A -85,B 0,C 180,E1 -26667.987,E2 -26667.987} C_VEL
LIN {X 0,Y 149.637,Z 432.915,A -85,B 0,C 180,E1 -26671.009,E2 -26671.009} C_VEL
LIN {X 0,Y 149.813,Z 448.735,A -85,B 0,C 180,E1 -26672.489,E2 -26672.489} C_VEL
LIN {X 0,Y 149.57,Z 467.779,A -85,B 0,C 180,E1 -26674.019,E2 -26674.019} C_VEL
LIN {X 0,Y 147.459,Z 481.043,A -85,B 0,C 180,E1 -26674.82,E2 -26674.82} C_VEL
LIN {X 0,Y 144.176,Z 493.984,A -85,B 0,C 180,E1 -26675.941,E2 -26675.941} C_VEL
LIN {X 0,Y 140.376,Z 505.416,A -85,B 0,C 180,E1 -26677.366,E2 -26677.366} C_VEL
LIN {X 0,Y 135.827,Z 516.093,A -85,B 0,C 180,E1 -26679.093,E2 -26679.093} C_VEL
LIN {X 0,Y 130.33,Z 527.058,A -85,B 0,C 180,E1 -26681.566,E2 -26681.566} C_VEL
LIN {X 0,Y 124.989,Z 536.004,A -85,B 0,C 180,E1 -26684.2,E2 -26684.2} C_VEL
LIN {X 0,Y 119.518,Z 544.267,A -85,B 0,C 180,E1 -26687.451,E2 -26687.451} C_VEL
LIN {X 0,Y 113.682,Z 552.43,A -85,B 0,C 180,E1 -26691.815,E2 -26691.815} C_VEL
LIN {X 0,Y 108.722,Z 559.034,A -85,B 0,C 180,E1 -26696.673,E2 -26696.673} C_VEL
LIN {X 0,Y 104.675,Z 564.323,A -85,B 0,C 180,E1 -26701.967,E2 -26701.967} C_VEL
LIN {X 0,Y 101.773,Z 568.505,A -85,B 0,C 180,E1 -26707.679,E2 -26707.679} C_VEL
LIN {X 0,Y 100.091,Z 571.678,A -85,B 0,C 180,E1 -26713.688,E2 -26713.688} C_VEL
LIN {X 0,Y 99.587,Z 574.394,A -85,B 0,C 180,E1 -26721.886,E2 -26721.886} C_VEL
LIN {X 0,Y 100.023,Z 575.158,A -85,B 0,C 180,E1 -26725.971,E2 -26725.971} C_VEL
LIN {X 0,Y 100.781,Z 575.504,A -85,B 0,C 180,E1 -26730,E2 -26730} C_VEL
LIN {X 0,Y 100.026,Z 575.141,A -85,B 0,C 180,E1 -26734.029,E2 -26734.029} C_VEL
LIN {X 0,Y 99.559,Z 574.209,A -85,B 0,C 180,E1 -26738.783,E2 -26738.783} C_VEL
LIN {X 0,Y 100.08,Z 571.62,A -85,B 0,C 180,E1 -26746.313,E2 -26746.313} C_VEL
LIN {X 0,Y 101.771,Z 568.425,A -85,B 0,C 180,E1 -26752.322,E2 -26752.322} C_VEL
LIN {X 0,Y 104.676,Z 564.215,A -85,B 0,C 180,E1 -26758.033,E2 -26758.033} C_VEL
LIN {X 0,Y 109.496,Z 557.856,A -85,B 0,C 180,E1 -26764.167,E2 -26764.167} C_VEL
LIN {X 0,Y 114.564,Z 550.976,A -85,B 0,C 180,E1 -26768.96,E2 -26768.96} C_VEL
LIN {X 0,Y 120.562,Z 542.528,A -85,B 0,C 180,E1 -26773.231,E2 -26773.231} C_VEL
LIN {X 0,Y 126.177,Z 533.91,A -85,B 0,C 180,E1 -26776.392,E2 -26776.392} C_VEL
LIN {X 0,Y 131.574,Z 524.487,A -85,B 0,C 180,E1 -26778.979,E2 -26778.979} C_VEL
LIN {X 0,Y 137.122,Z 512.799,A -85,B 0,C 180,E1 -26781.408,E2 -26781.408} C_VEL
LIN {X 0,Y 141.522,Z 501.71,A -85,B 0,C 180,E1 -26783.069,E2 -26783.069} C_VEL
LIN {X 0,Y 145.375,Z 488.929,A -85,B 0,C 180,E1 -26784.482,E2 -26784.482} C_VEL
LIN {X 0,Y 148.257,Z 475.483,A -85,B 0,C 180,E1 -26785.496,E2 -26785.496} C_VEL
LIN {X 0,Y 149.467,Z 466.196,A -85,B 0,C 180,E1 -26786.005,E2 -26786.005} C_VEL
LIN {X 0,Y 149.587,Z 457.692,A -85,B 0,C 180,E1 -26786.692,E2 -26786.692} C_VEL
LIN {X 0,Y 149.065,Z 450.089,A -85,B 0,C 180,E1 -26787.634,E2 -26787.634} C_VEL
LIN {X 0,Y 147.878,Z 442.958,A -85,B 0,C 180,E1 -26788.973,E2 -26788.973} C_VEL
LIN {X 0,Y 146.19,Z 436.399,A -85,B 0,C 180,E1 -26790.666,E2 -26790.666} C_VEL
LIN {X 0,Y 144.142,Z 430.534,A -85,B 0,C 180,E1 -26792.685,E2 -26792.685} C_VEL
LIN {X 0,Y 141.128,Z 421.186,A -85,B 0,C 180,E1 -26796.133,E2 -26796.133} C_VEL
LIN {X 0,Y 138.342,Z 413.675,A -85,B 0,C 180,E1 -26799.783,E2 -26799.783} C_VEL
LIN {X 0,Y 136.616,Z 409.42,A -85,B 0,C 180,E1 -26802.409,E2 -26802.409} C_VEL
LIN {X 0,Y 135.207,Z 405.83,A -85,B 0,C 180,E1 -26804.936,E2 -26804.936} C_VEL
LIN {X 0,Y 133.449,Z 401.598,A -85,B 0,C 180,E1 -26808.824,E2 -26808.824} C_VEL
LIN {X 0,Y 131.075,Z 396.884,A -85,B 0,C 180,E1 -26819.424,E2 -26819.424} C_VEL
LIN {X 0,Y 131.081,Z 397.121,A -85,B 0,C 180,E1 -26823.074,E2 -26823.074} C_VEL
LIN {X 0,Y 133.172,Z 401.448,A -85,B 0,C 180,E1 -26832.574,E2 -26832.574} C_VEL
LIN {X 0,Y 133.715,Z 402.345,A -85,B 0,C 180,E1 -26833.875,E2 -26833.875} C_VEL
LIN {X 0,Y 136.406,Z 406.725,A -85,B 0,C 180,E1 -26838.883,E2 -26838.883} C_VEL
LIN {X 0,Y 138.758,Z 410.572,A -85,B 0,C 180,E1 -26842.228,E2 -26842.228} C_VEL
LIN {X 0,Y 142.169,Z 416.506,A -85,B 0,C 180,E1 -26846.223,E2 -26846.223} C_VEL
LIN {X 0,Y 145.518,Z 423.024,A -85,B 0,C 180,E1 -26849.558,E2 -26849.558} C_VEL
LIN {X 0,Y 149.073,Z 430.658,A -85,B 0,C 180,E1 -26852.669,E2 -26852.669} C_VEL
LIN {X 0,Y 147.626,Z 448.256,A -85,B 0,C 180,E1 -26853.584,E2 -26853.584} C_VEL
LIN {X 0,Y 145.682,Z 460.356,A -85,B 0,C 180,E1 -26854.554,E2 -26854.554} C_VEL
LIN {X 0,Y 142.715,Z 472.728,A -85,B 0,C 180,E1 -26855.96,E2 -26855.96} C_VEL
LIN {X 0,Y 139.02,Z 483.964,A -85,B 0,C 180,E1 -26857.671,E2 -26857.671} C_VEL
LIN {X 0,Y 134.634,Z 494.318,A -85,B 0,C 180,E1 -26859.651,E2 -26859.651} C_VEL
LIN {X 0,Y 129.958,Z 503.59,A -85,B 0,C 180,E1 -26861.963,E2 -26861.963} C_VEL
LIN {X 0,Y 124.584,Z 513.026,A -85,B 0,C 180,E1 -26865.16,E2 -26865.16} C_VEL
LIN {X 0,Y 119.452,Z 520.755,A -85,B 0,C 180,E1 -26868.556,E2 -26868.556} C_VEL
LIN {X 0,Y 113.708,Z 528.403,A -85,B 0,C 180,E1 -26873.054,E2 -26873.054} C_VEL
LIN {X 0,Y 107.987,Z 535.199,A -85,B 0,C 180,E1 -26878.624,E2 -26878.624} C_VEL
LIN {X 0,Y 103.674,Z 539.802,A -85,B 0,C 180,E1 -26883.856,E2 -26883.856} C_VEL
LIN {X 0,Y 99.948,Z 543.349,A -85,B 0,C 180,E1 -26889.416,E2 -26889.416} C_VEL
LIN {X 0,Y 98.022,Z 545.17,A -85,B 0,C 180,E1 -26893.334,E2 -26893.334} C_VEL
LIN {X 0,Y 96.786,Z 546.496,A -85,B 0,C 180,E1 -26897.418,E2 -26897.418} C_VEL
LIN {X 0,Y 95.224,Z 548.037,A -85,B 0,C 180,E1 -26905.768,E2 -26905.768} C_VEL
LIN {X 0,Y 95.025,Z 548.257,A -85,B 0,C 180,E1 -26910,E2 -26910} C_VEL
LIN {X 0,Y 95.223,Z 548.065,A -85,B 0,C 180,E1 -26914.233,E2 -26914.233} C_VEL
LIN {X 0,Y 96.777,Z 546.559,A -85,B 0,C 180,E1 -26922.583,E2 -26922.583} C_VEL
LIN {X 0,Y 98.003,Z 545.263,A -85,B 0,C 180,E1 -26926.669,E2 -26926.669} C_VEL
LIN {X 0,Y 101.199,Z 542.412,A -85,B 0,C 180,E1 -26932.455,E2 -26932.455} C_VEL
LIN {X 0,Y 105.083,Z 538.574,A -85,B 0,C 180,E1 -26937.915,E2 -26937.915} C_VEL
LIN {X 0,Y 109.635,Z 533.481,A -85,B 0,C 180,E1 -26943.234,E2 -26943.234} C_VEL
LIN {X 0,Y 115.649,Z 526.226,A -85,B 0,C 180,E1 -26948.527,E2 -26948.527} C_VEL
LIN {X 0,Y 121.503,Z 518.187,A -85,B 0,C 180,E1 -26952.815,E2 -26952.815} C_VEL
LIN {X 0,Y 126.683,Z 509.95,A -85,B 0,C 180,E1 -26956.153,E2 -26956.153} C_VEL
LIN {X 0,Y 131.63,Z 500.894,A -85,B 0,C 180,E1 -26958.951,E2 -26958.951} C_VEL
LIN {X 0,Y 136.704,Z 490.335,A -85,B 0,C 180,E1 -26961.302,E2 -26961.302} C_VEL
LIN {X 0,Y 141.135,Z 478.623,A -85,B 0,C 180,E1 -26963.352,E2 -26963.352} C_VEL
LIN {X 0,Y 144.566,Z 467.098,A -85,B 0,C 180,E1 -26964.816,E2 -26964.816} C_VEL
LIN {X 0,Y 146.887,Z 455.215,A -85,B 0,C 180,E1 -26966.045,E2 -26966.045} C_VEL
LIN {X 0,Y 148.502,Z 442.4,A -85,B 0,C 180,E1 -26966.893,E2 -26966.893} C_VEL
LIN {X 0,Y 149.154,Z 430.567,A -85,B 0,C 180,E1 -26967.589,E2 -26967.589} C_VEL
LIN {X 0,Y 145.414,Z 422.548,A -85,B 0,C 180,E1 -26970.9,E2 -26970.9} C_VEL
LIN {X 0,Y 141.913,Z 415.855,A -85,B 0,C 180,E1 -26974.453,E2 -26974.453} C_VEL
LIN {X 0,Y 139.212,Z 411.125,A -85,B 0,C 180,E1 -26977.653,E2 -26977.653} C_VEL
LIN {X 0,Y 137.498,Z 408.433,A -85,B 0,C 180,E1 -26979.975,E2 -26979.975} C_VEL
LIN {X 0,Y 135.905,Z 405.741,A -85,B 0,C 180,E1 -26982.507,E2 -26982.507} C_VEL
LIN {X 0,Y 133.487,Z 401.634,A -85,B 0,C 180,E1 -26987.501,E2 -26987.501} C_VEL
LIN {X 0,Y 131.335,Z 397.191,A -85,B 0,C 180,E1 -26998.735,E2 -26998.735} C_VEL
LIN {X 0,Y 131.36,Z 397.227,A -85,B 0,C 180,E1 -27000.287,E2 -27000.287} C_VEL
LIN {X 0,Y 133.73,Z 401.987,A -85,B 0,C 180,E1 -27011.174,E2 -27011.174} C_VEL
LIN {X 0,Y 136.104,Z 407.582,A -85,B 0,C 180,E1 -27016.186,E2 -27016.186} C_VEL
LIN {X 0,Y 138.376,Z 413.365,A -85,B 0,C 180,E1 -27019.856,E2 -27019.856} C_VEL
LIN {X 0,Y 141.088,Z 420.713,A -85,B 0,C 180,E1 -27023.485,E2 -27023.485} C_VEL
LIN {X 0,Y 144.019,Z 429.578,A -85,B 0,C 180,E1 -27026.878,E2 -27026.878} C_VEL
LIN {X 0,Y 145.987,Z 436.217,A -85,B 0,C 180,E1 -27028.955,E2 -27028.955} C_VEL
LIN {X 0,Y 145.824,Z 462.477,A -85,B 0,C 180,E1 -27031.31,E2 -27031.31} C_VEL
LIN {X 0,Y 145.376,Z 469.352,A -85,B 0,C 180,E1 -27031.832,E2 -27031.832} C_VEL
LIN {X 0,Y 142.781,Z 483.187,A -85,B 0,C 180,E1 -27032.695,E2 -27032.695} C_VEL
LIN {X 0,Y 139.757,Z 494.16,A -85,B 0,C 180,E1 -27033.695,E2 -27033.695} C_VEL
LIN {X 0,Y 135.504,Z 506.108,A -85,B 0,C 180,E1 -27035.227,E2 -27035.227} C_VEL
LIN {X 0,Y 130.135,Z 517.721,A -85,B 0,C 180,E1 -27037.197,E2 -27037.197} C_VEL
LIN {X 0,Y 125.092,Z 527.151,A -85,B 0,C 180,E1 -27039.421,E2 -27039.421} C_VEL
LIN {X 0,Y 118.934,Z 536.819,A -85,B 0,C 180,E1 -27042.385,E2 -27042.385} C_VEL
LIN {X 0,Y 113.286,Z 544.79,A -85,B 0,C 180,E1 -27045.74,E2 -27045.74} C_VEL
LIN {X 0,Y 107.197,Z 552.622,A -85,B 0,C 180,E1 -27050.267,E2 -27050.267} C_VEL
LIN {X 0,Y 101.267,Z 559.923,A -85,B 0,C 180,E1 -27056.276,E2 -27056.276} C_VEL
LIN {X 0,Y 97.195,Z 564.828,A -85,B 0,C 180,E1 -27061.966,E2 -27061.966} C_VEL
LIN {X 0,Y 94.37,Z 568.656,A -85,B 0,C 180,E1 -27068.139,E2 -27068.139} C_VEL
LIN {X 0,Y 93.221,Z 570.679,A -85,B 0,C 180,E1 -27072.449,E2 -27072.449} C_VEL
LIN {X 0,Y 92.526,Z 573.401,A -85,B 0,C 180,E1 -27081.262,E2 -27081.262} C_VEL
LIN {X 0,Y 92.914,Z 574.166,A -85,B 0,C 180,E1 -27085.662,E2 -27085.662} C_VEL
LIN {X 0,Y 93.673,Z 574.515,A -85,B 0,C 180,E1 -27090,E2 -27090} C_VEL
LIN {X 0,Y 92.917,Z 574.149,A -85,B 0,C 180,E1 -27094.338,E2 -27094.338} C_VEL
LIN {X 0,Y 92.494,Z 573.32,A -85,B 0,C 180,E1 -27098.964,E2 -27098.964} C_VEL
LIN {X 0,Y 93.211,Z 570.62,A -85,B 0,C 180,E1 -27107.553,E2 -27107.553} C_VEL
LIN {X 0,Y 95.168,Z 567.425,A -85,B 0,C 180,E1 -27113.964,E2 -27113.964} C_VEL
LIN {X 0,Y 99.316,Z 562.159,A -85,B 0,C 180,E1 -27121.204,E2 -27121.204} C_VEL
LIN {X 0,Y 104.49,Z 555.814,A -85,B 0,C 180,E1 -27127.252,E2 -27127.252} C_VEL
LIN {X 0,Y 110.153,Z 548.727,A -85,B 0,C 180,E1 -27132.06,E2 -27132.06} C_VEL
LIN {X 0,Y 116.611,Z 539.911,A -85,B 0,C 180,E1 -27136.32,E2 -27136.32} C_VEL
LIN {X 0,Y 122.572,Z 530.939,A -85,B 0,C 180,E1 -27139.439,E2 -27139.439} C_VEL
LIN {X 0,Y 128.26,Z 521.116,A -85,B 0,C 180,E1 -27141.967,E2 -27141.967} C_VEL
LIN {X 0,Y 133.478,Z 510.364,A -85,B 0,C 180,E1 -27144.049,E2 -27144.049} C_VEL
LIN {X 0,Y 138.227,Z 498.304,A -85,B 0,C 180,E1 -27145.723,E2 -27145.723} C_VEL
LIN {X 0,Y 141.967,Z 485.642,A -85,B 0,C 180,E1 -27147.024,E2 -27147.024} C_VEL
LIN {X 0,Y 144.674,Z 472.621,A -85,B 0,C 180,E1 -27147.933,E2 -27147.933} C_VEL
LIN {X 0,Y 145.428,Z 466.65,A -85,B 0,C 180,E1 -27148.282,E2 -27148.282} C_VEL
LIN {X 0,Y 145.778,Z 438.598,A -85,B 0,C 180,E1 -27150.732,E2 -27150.732} C_VEL
LIN {X 0,Y 145.689,Z 435.733,A -85,B 0,C 180,E1 -27151.069,E2 -27151.069} C_VEL
LIN {X 0,Y 144.142,Z 430.534,A -85,B 0,C 180,E1 -27152.685,E2 -27152.685} C_VEL
LIN {X 0,Y 142.883,Z 428.269,A -85,B 0,C 180,E1 -27153.88,E2 -27153.88} C_VEL
LIN {X 0,Y 140.438,Z 425.827,A -85,B 0,C 180,E1 -27156.188,E2 -27156.188} C_VEL
LIN {X 0,Y 137.732,Z 423.069,A -85,B 0,C 180,E1 -27159.121,E2 -27159.121} C_VEL
LIN {X 0,Y 137.041,Z 421.719,A -85,B 0,C 180,E1 -27160.045,E2 -27160.045} C_VEL
LIN {X 0,Y 135.38,Z 417.011,A -85,B 0,C 180,E1 -27162.73,E2 -27162.73} C_VEL
LIN {X 0,Y 133.63,Z 412.178,A -85,B 0,C 180,E1 -27166.12,E2 -27166.12} C_VEL
LIN {X 0,Y 132.228,Z 408.464,A -85,B 0,C 180,E1 -27169.566,E2 -27169.566} C_VEL
LIN {X 0,Y 130.19,Z 403.843,A -85,B 0,C 180,E1 -27180,E2 -27180} C_VEL
LIN {X 0,Y 130.202,Z 404.295,A -85,B 0,C 180,E1 -27183.094,E2 -27183.094} C_VEL
LIN {X 0,Y 132.158,Z 408.445,A -85,B 0,C 180,E1 -27192.282,E2 -27192.282} C_VEL
LIN {X 0,Y 134.848,Z 413.304,A -85,B 0,C 180,E1 -27197.924,E2 -27197.924} C_VEL
LIN {X 0,Y 137.194,Z 417.43,A -85,B 0,C 180,E1 -27201.506,E2 -27201.506} C_VEL
LIN {X 0,Y 140.121,Z 422.877,A -85,B 0,C 180,E1 -27205.176,E2 -27205.176} C_VEL
LIN {X 0,Y 143.37,Z 429.661,A -85,B 0,C 180,E1 -27208.648,E2 -27208.648} C_VEL
LIN {X 0,Y 145.216,Z 433.805,A -85,B 0,C 180,E1 -27210.42,E2 -27210.42} C_VEL
LIN {X 0,Y 143.715,Z 450.265,A -85,B 0,C 180,E1 -27211.31,E2 -27211.31} C_VEL
LIN {X 0,Y 141.454,Z 463.046,A -85,B 0,C 180,E1 -27212.37,E2 -27212.37} C_VEL
LIN {X 0,Y 138.397,Z 474.694,A -85,B 0,C 180,E1 -27213.747,E2 -27213.747} C_VEL
LIN {X 0,Y 134.118,Z 486.795,A -85,B 0,C 180,E1 -27215.64,E2 -27215.64} C_VEL
LIN {X 0,Y 129.65,Z 496.571,A -85,B 0,C 180,E1 -27217.555,E2 -27217.555} C_VEL
LIN {X 0,Y 124.805,Z 505.616,A -85,B 0,C 180,E1 -27219.894,E2 -27219.894} C_VEL
LIN {X 0,Y 119.702,Z 514.007,A -85,B 0,C 180,E1 -27222.787,E2 -27222.787} C_VEL
LIN {X 0,Y 114.278,Z 521.736,A -85,B 0,C 180,E1 -27226.223,E2 -27226.223} C_VEL
LIN {X 0,Y 108.173,Z 529.383,A -85,B 0,C 180,E1 -27230.816,E2 -27230.816} C_VEL
LIN {X 0,Y 102.052,Z 536.178,A -85,B 0,C 180,E1 -27236.57,E2 -27236.57} C_VEL
LIN {X 0,Y 97.414,Z 540.781,A -85,B 0,C 180,E1 -27242.035,E2 -27242.035} C_VEL
LIN {X 0,Y 93.399,Z 544.328,A -85,B 0,C 180,E1 -27247.9,E2 -27247.9} C_VEL
LIN {X 0,Y 91.308,Z 546.149,A -85,B 0,C 180,E1 -27252.069,E2 -27252.069} C_VEL
LIN {X 0,Y 89.938,Z 547.475,A -85,B 0,C 180,E1 -27256.442,E2 -27256.442} C_VEL
LIN {X 0,Y 88.216,Z 549.015,A -85,B 0,C 180,E1 -27265.431,E2 -27265.431} C_VEL
LIN {X 0,Y 87.997,Z 549.235,A -85,B 0,C 180,E1 -27270,E2 -27270} C_VEL
LIN {X 0,Y 88.216,Z 549.043,A -85,B 0,C 180,E1 -27274.569,E2 -27274.569} C_VEL
LIN {X 0,Y 89.929,Z 547.537,A -85,B 0,C 180,E1 -27283.559,E2 -27283.559} C_VEL
LIN {X 0,Y 91.289,Z 546.241,A -85,B 0,C 180,E1 -27287.935,E2 -27287.935} C_VEL
LIN {X 0,Y 94.742,Z 543.389,A -85,B 0,C 180,E1 -27294.078,E2 -27294.078} C_VEL
LIN {X 0,Y 98.927,Z 539.551,A -85,B 0,C 180,E1 -27299.821,E2 -27299.821} C_VEL
LIN {X 0,Y 103.828,Z 534.458,A -85,B 0,C 180,E1 -27305.36,E2 -27305.36} C_VEL
LIN {X 0,Y 110.238,Z 527.202,A -85,B 0,C 180,E1 -27310.803,E2 -27310.803} C_VEL
LIN {X 0,Y 116.445,Z 519.162,A -85,B 0,C 180,E1 -27315.166,E2 -27315.166} C_VEL
LIN {X 0,Y 121.918,Z 510.926,A -85,B 0,C 180,E1 -27318.536,E2 -27318.536} C_VEL
LIN {X 0,Y 127.122,Z 501.869,A -85,B 0,C 180,E1 -27321.343,E2 -27321.343} C_VEL
LIN {X 0,Y 132.426,Z 491.307,A -85,B 0,C 180,E1 -27323.676,E2 -27323.676} C_VEL
LIN {X 0,Y 136.993,Z 479.752,A -85,B 0,C 180,E1 -27325.69,E2 -27325.69} C_VEL
LIN {X 0,Y 140.531,Z 468.42,A -85,B 0,C 180,E1 -27327.124,E2 -27327.124} C_VEL
LIN {X 0,Y 143.173,Z 455.619,A -85,B 0,C 180,E1 -27328.424,E2 -27328.424} C_VEL
LIN {X 0,Y 144.864,Z 442.229,A -85,B 0,C 180,E1 -27329.299,E2 -27329.299} C_VEL
LIN {X 0,Y 145.389,Z 433.908,A -85,B 0,C 180,E1 -27329.773,E2 -27329.773} C_VEL
LIN {X 0,Y 141.54,Z 425.427,A -85,B 0,C 180,E1 -27333.652,E2 -27333.652} C_VEL
LIN {X 0,Y 138.076,Z 418.663,A -85,B 0,C 180,E1 -27337.804,E2 -27337.804} C_VEL
LIN {X 0,Y 135.965,Z 415.077,A -85,B 0,C 180,E1 -27340.809,E2 -27340.809} C_VEL
LIN {X 0,Y 134.406,Z 412.281,A -85,B 0,C 180,E1 -27343.484,E2 -27343.484} C_VEL
LIN {X 0,Y 132.265,Z 408.445,A -85,B 0,C 180,E1 -27348.312,E2 -27348.312} C_VEL
LIN {X 0,Y 130.467,Z 404.264,A -85,B 0,C 180,E1 -27358.727,E2 -27358.727} C_VEL
LIN {X 0,Y 130.475,Z 404.56,A -85,B 0,C 180,E1 -27360.579,E2 -27360.579} C_VEL
LIN {X 0,Y 132.473,Z 408.719,A -85,B 0,C 180,E1 -27370.314,E2 -27370.314} C_VEL
LIN {X 0,Y 134.349,Z 413.614,A -85,B 0,C 180,E1 -27374.775,E2 -27374.775} C_VEL
LIN {X 0,Y 136.39,Z 419.408,A -85,B 0,C 180,E1 -27378.495,E2 -27378.495} C_VEL
LIN {X 0,Y 138.613,Z 426.002,A -85,B 0,C 180,E1 -27381.83,E2 -27381.83} C_VEL
LIN {X 0,Y 141.079,Z 434.179,A -85,B 0,C 180,E1 -27385.052,E2 -27385.052} C_VEL
LIN {X 0,Y 142.493,Z 439.678,A -85,B 0,C 180,E1 -27386.783,E2 -27386.783} C_VEL
LIN {X 0,Y 141.917,Z 466.316,A -85,B 0,C 180,E1 -27389.193,E2 -27389.193} C_VEL
LIN {X 0,Y 140.34,Z 476.432,A -85,B 0,C 180,E1 -27389.82,E2 -27389.82} C_VEL
LIN {X 0,Y 137.356,Z 488.686,A -85,B 0,C 180,E1 -27390.775,E2 -27390.775} C_VEL
LIN {X 0,Y 133.527,Z 500.058,A -85,B 0,C 180,E1 -27391.998,E2 -27391.998} C_VEL
LIN {X 0,Y 128.76,Z 511.274,A -85,B 0,C 180,E1 -27393.657,E2 -27393.657} C_VEL
LIN {X 0,Y 123.283,Z 521.67,A -85,B 0,C 180,E1 -27395.675,E2 -27395.675} C_VEL
LIN {X 0,Y 118.07,Z 530.256,A -85,B 0,C 180,E1 -27397.938,E2 -27397.938} C_VEL
LIN {X 0,Y 111.804,Z 539.173,A -85,B 0,C 180,E1 -27401.035,E2 -27401.035} C_VEL
LIN {X 0,Y 104.984,Z 547.93,A -85,B 0,C 180,E1 -27405.34,E2 -27405.34} C_VEL
LIN {X 0,Y 98.902,Z 554.976,A -85,B 0,C 180,E1 -27410.243,E2 -27410.243} C_VEL
LIN {X 0,Y 93.905,Z 560.566,A -85,B 0,C 180,E1 -27415.672,E2 -27415.672} C_VEL
LIN {X 0,Y 89.736,Z 565.214,A -85,B 0,C 180,E1 -27421.972,E2 -27421.972} C_VEL
LIN {X 0,Y 87.005,Z 568.708,A -85,B 0,C 180,E1 -27428.685,E2 -27428.685} C_VEL
LIN {X 0,Y 85.608,Z 571.237,A -85,B 0,C 180,E1 -27435.742,E2 -27435.742} C_VEL
LIN {X 0,Y 85.812,Z 573.175,A -85,B 0,C 180,E1 -27445.302,E2 -27445.302} C_VEL
LIN {X 0,Y 86.561,Z 573.526,A -85,B 0,C 180,E1 -27450,E2 -27450} C_VEL
LIN {X 0,Y 85.814,Z 573.158,A -85,B 0,C 180,E1 -27454.698,E2 -27454.698} C_VEL
LIN {X 0,Y 85.604,Z 571.197,A -85,B 0,C 180,E1 -27464.258,E2 -27464.258} C_VEL
LIN {X 0,Y 86.997,Z 568.642,A -85,B 0,C 180,E1 -27471.317,E2 -27471.317} C_VEL
LIN {X 0,Y 89.74,Z 565.119,A -85,B 0,C 180,E1 -27478.026,E2 -27478.026} C_VEL
LIN {X 0,Y 94.59,Z 559.692,A -85,B 0,C 180,E1 -27485.185,E2 -27485.185} C_VEL
LIN {X 0,Y 99.835,Z 553.753,A -85,B 0,C 180,E1 -27490.628,E2 -27490.628} C_VEL
LIN {X 0,Y 106.069,Z 546.372,A -85,B 0,C 180,E1 -27495.42,E2 -27495.42} C_VEL
LIN {X 0,Y 113.02,Z 537.265,A -85,B 0,C 180,E1 -27499.617,E2 -27499.617} C_VEL
LIN {X 0,Y 119.376,Z 527.967,A -85,B 0,C 180,E1 -27502.633,E2 -27502.633} C_VEL
LIN {X 0,Y 124.646,Z 518.921,A -85,B 0,C 180,E1 -27504.84,E2 -27504.84} C_VEL
LIN {X 0,Y 130.113,Z 507.794,A -85,B 0,C 180,E1 -27506.846,E2 -27506.846} C_VEL
LIN {X 0,Y 134.981,Z 495.385,A -85,B 0,C 180,E1 -27508.476,E2 -27508.476} C_VEL
LIN {X 0,Y 138.523,Z 483.517,A -85,B 0,C 180,E1 -27509.597,E2 -27509.597} C_VEL
LIN {X 0,Y 141.249,Z 470.268,A -85,B 0,C 180,E1 -27510.437,E2 -27510.437} C_VEL
LIN {X 0,Y 141.92,Z 459.712,A -85,B 0,C 180,E1 -27511.33,E2 -27511.33} C_VEL
LIN {X 0,Y 142.25,Z 439.048,A -85,B 0,C 180,E1 -27513.216,E2 -27513.216} C_VEL
LIN {X 0,Y 139.416,Z 429.087,A -85,B 0,C 180,E1 -27516.709,E2 -27516.709} C_VEL
LIN {X 0,Y 137.041,Z 421.719,A -85,B 0,C 180,E1 -27520.045,E2 -27520.045} C_VEL
LIN {X 0,Y 135.581,Z 418.955,A -85,B 0,C 180,E1 -27522.159,E2 -27522.159} C_VEL
LIN {X 0,Y 134.062,Z 417.189,A -85,B 0,C 180,E1 -27524.488,E2 -27524.488} C_VEL
LIN {X 0,Y 130.169,Z 414.156,A -85,B 0,C 180,E1 -27533.009,E2 -27533.009} C_VEL
LIN {X 0,Y 129.321,Z 410.925,A -85,B 0,C 180,E1 -27540,E2 -27540} C_VEL
LIN {X 0,Y 129.315,Z 411.293,A -85,B 0,C 180,E1 -27542.726,E2 -27542.726} C_VEL
LIN {X 0,Y 131.16,Z 415.696,A -85,B 0,C 180,E1 -27552.082,E2 -27552.082} C_VEL
LIN {X 0,Y 133.373,Z 419.956,A -85,B 0,C 180,E1 -27557.023,E2 -27557.023} C_VEL
LIN {X 0,Y 135.355,Z 423.68,A -85,B 0,C 180,E1 -27560.318,E2 -27560.318} C_VEL
LIN {X 0,Y 138.123,Z 429.21,A -85,B 0,C 180,E1 -27564.094,E2 -27564.094} C_VEL
LIN {X 0,Y 141.266,Z 436.361,A -85,B 0,C 180,E1 -27567.724,E2 -27567.724} C_VEL
LIN {X 0,Y 141.578,Z 437.112,A -85,B 0,C 180,E1 -27568.056,E2 -27568.056} C_VEL
LIN {X 0,Y 140.04,Z 452.522,A -85,B 0,C 180,E1 -27568.952,E2 -27568.952} C_VEL
LIN {X 0,Y 137.503,Z 465.218,A -85,B 0,C 180,E1 -27570.007,E2 -27570.007} C_VEL
LIN {X 0,Y 133.823,Z 478.077,A -85,B 0,C 180,E1 -27571.581,E2 -27571.581} C_VEL
LIN {X 0,Y 129.444,Z 489.428,A -85,B 0,C 180,E1 -27573.403,E2 -27573.403} C_VEL
LIN {X 0,Y 124.848,Z 498.817,A -85,B 0,C 180,E1 -27575.291,E2 -27575.291} C_VEL
LIN {X 0,Y 119.808,Z 507.638,A -85,B 0,C 180,E1 -27577.637,E2 -27577.637} C_VEL
LIN {X 0,Y 113.893,Z 516.646,A -85,B 0,C 180,E1 -27580.896,E2 -27580.896} C_VEL
LIN {X 0,Y 107.131,Z 525.397,A -85,B 0,C 180,E1 -27585.154,E2 -27585.154} C_VEL
LIN {X 0,Y 101.715,Z 531.559,A -85,B 0,C 180,E1 -27589.237,E2 -27589.237} C_VEL
LIN {X 0,Y 96.265,Z 537.158,A -85,B 0,C 180,E1 -27594.265,E2 -27594.265} C_VEL
LIN {X 0,Y 91.266,Z 541.76,A -85,B 0,C 180,E1 -27599.965,E2 -27599.965} C_VEL
LIN {X 0,Y 86.924,Z 545.307,A -85,B 0,C 180,E1 -27606.156,E2 -27606.156} C_VEL
LIN {X 0,Y 84.646,Z 547.128,A -85,B 0,C 180,E1 -27610.603,E2 -27610.603} C_VEL
LIN {X 0,Y 83.12,Z 548.453,A -85,B 0,C 180,E1 -27615.306,E2 -27615.306} C_VEL
LIN {X 0,Y 81.212,Z 549.994,A -85,B 0,C 180,E1 -27625.036,E2 -27625.036} C_VEL
LIN {X 0,Y 80.969,Z 550.213,A -85,B 0,C 180,E1 -27630,E2 -27630} C_VEL
LIN {X 0,Y 81.212,Z 550.02,A -85,B 0,C 180,E1 -27634.965,E2 -27634.965} C_VEL
LIN {X 0,Y 83.111,Z 548.515,A -85,B 0,C 180,E1 -27644.695,E2 -27644.695} C_VEL
LIN {X 0,Y 84.627,Z 547.219,A -85,B 0,C 180,E1 -27649.401,E2 -27649.401} C_VEL
LIN {X 0,Y 88.372,Z 544.366,A -85,B 0,C 180,E1 -27655.938,E2 -27655.938} C_VEL
LIN {X 0,Y 92.895,Z 540.528,A -85,B 0,C 180,E1 -27661.977,E2 -27661.977} C_VEL
LIN {X 0,Y 98.181,Z 535.434,A -85,B 0,C 180,E1 -27667.734,E2 -27667.734} C_VEL
LIN {X 0,Y 105.019,Z 528.178,A -85,B 0,C 180,E1 -27673.309,E2 -27673.309} C_VEL
LIN {X 0,Y 111.6,Z 520.138,A -85,B 0,C 180,E1 -27677.726,E2 -27677.726} C_VEL
LIN {X 0,Y 117.381,Z 511.901,A -85,B 0,C 180,E1 -27681.109,E2 -27681.109} C_VEL
LIN {X 0,Y 122.852,Z 502.844,A -85,B 0,C 180,E1 -27683.905,E2 -27683.905} C_VEL
LIN {X 0,Y 128.389,Z 492.28,A -85,B 0,C 180,E1 -27686.203,E2 -27686.203} C_VEL
LIN {X 0,Y 133.158,Z 480.724,A -85,B 0,C 180,E1 -27688.189,E2 -27688.189} C_VEL
LIN {X 0,Y 136.844,Z 469.391,A -85,B 0,C 180,E1 -27689.595,E2 -27689.595} C_VEL
LIN {X 0,Y 139.524,Z 457.147,A -85,B 0,C 180,E1 -27690.838,E2 -27690.838} C_VEL
LIN {X 0,Y 141.285,Z 444.465,A -85,B 0,C 180,E1 -27691.678,E2 -27691.678} C_VEL
LIN {X 0,Y 141.777,Z 437.213,A -85,B 0,C 180,E1 -27692.129,E2 -27692.129} C_VEL
LIN {X 0,Y 138.706,Z 430.184,A -85,B 0,C 180,E1 -27695.628,E2 -27695.628} C_VEL
LIN {X 0,Y 135.816,Z 424.25,A -85,B 0,C 180,E1 -27699.526,E2 -27699.526} C_VEL
LIN {X 0,Y 133.237,Z 419.258,A -85,B 0,C 180,E1 -27703.923,E2 -27703.923} C_VEL
LIN {X 0,Y 131.056,Z 415.223,A -85,B 0,C 180,E1 -27709.182,E2 -27709.182} C_VEL
LIN {X 0,Y 129.595,Z 411.367,A -85,B 0,C 180,E1 -27718.718,E2 -27718.718} C_VEL
LIN {X 0,Y 129.597,Z 411.868,A -85,B 0,C 180,E1 -27720.874,E2 -27720.874} C_VEL
LIN {X 0,Y 131.309,Z 415.582,A -85,B 0,C 180,E1 -27729.628,E2 -27729.628} C_VEL
LIN {X 0,Y 132.781,Z 420.042,A -85,B 0,C 180,E1 -27733.584,E2 -27733.584} C_VEL
LIN {X 0,Y 134.417,Z 425.234,A -85,B 0,C 180,E1 -27736.972,E2 -27736.972} C_VEL
LIN {X 0,Y 136.467,Z 431.981,A -85,B 0,C 180,E1 -27740.44,E2 -27740.44} C_VEL
LIN {X 0,Y 138.887,Z 441.115,A -85,B 0,C 180,E1 -27743.979,E2 -27743.979} C_VEL
LIN {X 0,Y 139.202,Z 442.897,A -85,B 0,C 180,E1 -27744.467,E2 -27744.467} C_VEL
LIN {X 0,Y 138.343,Z 466.86,A -85,B 0,C 180,E1 -27746.686,E2 -27746.686} C_VEL
LIN {X 0,Y 137.328,Z 473.56,A -85,B 0,C 180,E1 -27747.137,E2 -27747.137} C_VEL
LIN {X 0,Y 134.097,Z 486.828,A -85,B 0,C 180,E1 -27748.074,E2 -27748.074} C_VEL
LIN {X 0,Y 129.827,Z 499.238,A -85,B 0,C 180,E1 -27749.354,E2 -27749.354} C_VEL
LIN {X 0,Y 124.245,Z 511.725,A -85,B 0,C 180,E1 -27751.181,E2 -27751.181} C_VEL
LIN {X 0,Y 118.577,Z 521.868,A -85,B 0,C 180,E1 -27753.158,E2 -27753.158} C_VEL
LIN {X 0,Y 112.501,Z 531.233,A -85,B 0,C 180,E1 -27755.698,E2 -27755.698} C_VEL
LIN {X 0,Y 106.011,Z 539.787,A -85,B 0,C 180,E1 -27758.835,E2 -27758.835} C_VEL
LIN {X 0,Y 98.885,Z 548.198,A -85,B 0,C 180,E1 -27763.241,E2 -27763.241} C_VEL
LIN {X 0,Y 92.53,Z 555.026,A -85,B 0,C 180,E1 -27768.349,E2 -27768.349} C_VEL
LIN {X 0,Y 86.362,Z 561.346,A -85,B 0,C 180,E1 -27775.275,E2 -27775.275} C_VEL
LIN {X 0,Y 82.283,Z 565.514,A -85,B 0,C 180,E1 -27781.981,E2 -27781.981} C_VEL
LIN {X 0,Y 79.66,Z 568.684,A -85,B 0,C 180,E1 -27789.335,E2 -27789.335} C_VEL
LIN {X 0,Y 78.363,Z 571.403,A -85,B 0,C 180,E1 -27799.667,E2 -27799.667} C_VEL
LIN {X 0,Y 78.685,Z 572.18,A -85,B 0,C 180,E1 -27804.876,E2 -27804.876} C_VEL
LIN {X 0,Y 79.448,Z 572.536,A -85,B 0,C 180,E1 -27810,E2 -27810} C_VEL
LIN {X 0,Y 78.388,Z 571.528,A -85,B 0,C 180,E1 -27819.523,E2 -27819.523} C_VEL
LIN {X 0,Y 78.675,Z 570.199,A -85,B 0,C 180,E1 -27825.544,E2 -27825.544} C_VEL
LIN {X 0,Y 80.337,Z 567.64,A -85,B 0,C 180,E1 -27833.182,E2 -27833.182} C_VEL
LIN {X 0,Y 83.495,Z 564.123,A -85,B 0,C 180,E1 -27840.333,E2 -27840.333} C_VEL
LIN {X 0,Y 88.41,Z 559.113,A -85,B 0,C 180,E1 -27847.351,E2 -27847.351} C_VEL
LIN {X 0,Y 94.516,Z 552.755,A -85,B 0,C 180,E1 -27853.456,E2 -27853.456} C_VEL
LIN {X 0,Y 101.191,Z 545.378,A -85,B 0,C 180,E1 -27858.297,E2 -27858.297} C_VEL
LIN {X 0,Y 108.548,Z 536.272,A -85,B 0,C 180,E1 -27862.478,E2 -27862.478} C_VEL
LIN {X 0,Y 115.211,Z 526.977,A -85,B 0,C 180,E1 -27865.436,E2 -27865.436} C_VEL
LIN {X 0,Y 120.686,Z 517.927,A -85,B 0,C 180,E1 -27867.605,E2 -27867.605} C_VEL
LIN {X 0,Y 126.361,Z 506.798,A -85,B 0,C 180,E1 -27869.549,E2 -27869.549} C_VEL
LIN {X 0,Y 131.22,Z 494.881,A -85,B 0,C 180,E1 -27871.069,E2 -27871.069} C_VEL
LIN {X 0,Y 135.063,Z 482.518,A -85,B 0,C 180,E1 -27872.2,E2 -27872.2} C_VEL
LIN {X 0,Y 137.8,Z 469.772,A -85,B 0,C 180,E1 -27872.984,E2 -27872.984} C_VEL
LIN {X 0,Y 138.657,Z 454.032,A -85,B 0,C 180,E1 -27874.428,E2 -27874.428} C_VEL
LIN {X 0,Y 138.935,Z 442.066,A -85,B 0,C 180,E1 -27875.576,E2 -27875.576} C_VEL
LIN {X 0,Y 136.44,Z 432.564,A -85,B 0,C 180,E1 -27879.159,E2 -27879.159} C_VEL
LIN {X 0,Y 134.273,Z 425.275,A -85,B 0,C 180,E1 -27882.779,E2 -27882.779} C_VEL
LIN {X 0,Y 132.336,Z 419.103,A -85,B 0,C 180,E1 -27886.809,E2 -27886.809} C_VEL
LIN {X 0,Y 131.025,Z 415.274,A -85,B 0,C 180,E1 -27890.351,E2 -27890.351} C_VEL
LIN {X 0,Y 130.169,Z 414.156,A -85,B 0,C 180,E1 -27893.009,E2 -27893.009} C_VEL
LIN {X 0,Y 129.704,Z 413.958,A -85,B 0,C 180,E1 -27894.735,E2 -27894.735} C_VEL
LIN {X 0,Y 128.997,Z 415.253,A -85,B 0,C 180,E1 -27897.599,E2 -27897.599} C_VEL
LIN {X 0,Y 128.432,Z 418.253,A -85,B 0,C 180,E1 -27902.25,E2 -27902.25} C_VEL
LIN {X 0,Y 129.972,Z 422.527,A -85,B 0,C 180,E1 -27911.304,E2 -27911.304} C_VEL
LIN {X 0,Y 131.996,Z 426.744,A -85,B 0,C 180,E1 -27916.233,E2 -27916.233} C_VEL
LIN {X 0,Y 134.083,Z 430.97,A -85,B 0,C 180,E1 -27919.92,E2 -27919.92} C_VEL
LIN {X 0,Y 136.621,Z 436.581,A -85,B 0,C 180,E1 -27923.578,E2 -27923.578} C_VEL
LIN {X 0,Y 138.201,Z 440.546,A -85,B 0,C 180,E1 -27925.595,E2 -27925.595} C_VEL
LIN {X 0,Y 136.655,Z 454.189,A -85,B 0,C 180,E1 -27926.41,E2 -27926.41} C_VEL
LIN {X 0,Y 133.88,Z 467.167,A -85,B 0,C 180,E1 -27927.509,E2 -27927.509} C_VEL
LIN {X 0,Y 130.234,Z 479.212,A -85,B 0,C 180,E1 -27928.973,E2 -27928.973} C_VEL
LIN {X 0,Y 125.71,Z 490.416,A -85,B 0,C 180,E1 -27930.73,E2 -27930.73} C_VEL
LIN {X 0,Y 120.924,Z 499.798,A -85,B 0,C 180,E1 -27932.573,E2 -27932.573} C_VEL
LIN {X 0,Y 115.649,Z 508.62,A -85,B 0,C 180,E1 -27934.877,E2 -27934.877} C_VEL
LIN {X 0,Y 109.42,Z 517.626,A -85,B 0,C 180,E1 -27938.113,E2 -27938.113} C_VEL
LIN {X 0,Y 102.268,Z 526.378,A -85,B 0,C 180,E1 -27942.376,E2 -27942.376} C_VEL
LIN {X 0,Y 96.501,Z 532.538,A -85,B 0,C 180,E1 -27946.511,E2 -27946.511} C_VEL
LIN {X 0,Y 90.653,Z 538.137,A -85,B 0,C 180,E1 -27951.669,E2 -27951.669} C_VEL
LIN {X 0,Y 85.255,Z 542.74,A -85,B 0,C 180,E1 -27957.6,E2 -27957.6} C_VEL
LIN {X 0,Y 80.543,Z 546.287,A -85,B 0,C 180,E1 -27964.133,E2 -27964.133} C_VEL
LIN {X 0,Y 78.048,Z 548.107,A -85,B 0,C 180,E1 -27968.889,E2 -27968.889} C_VEL
LIN {X 0,Y 76.341,Z 549.432,A -85,B 0,C 180,E1 -27973.968,E2 -27973.968} C_VEL
LIN {X 0,Y 74.213,Z 550.972,A -85,B 0,C 180,E1 -27984.566,E2 -27984.566} C_VEL
LIN {X 0,Y 73.941,Z 551.191,A -85,B 0,C 180,E1 -27990,E2 -27990} C_VEL
LIN {X 0,Y 74.212,Z 550.998,A -85,B 0,C 180,E1 -27995.434,E2 -27995.434} C_VEL
LIN {X 0,Y 76.332,Z 549.493,A -85,B 0,C 180,E1 -28006.034,E2 -28006.034} C_VEL
LIN {X 0,Y 78.029,Z 548.196,A -85,B 0,C 180,E1 -28011.117,E2 -28011.117} C_VEL
LIN {X 0,Y 82.11,Z 545.343,A -85,B 0,C 180,E1 -28018.083,E2 -28018.083} C_VEL
LIN {X 0,Y 87.013,Z 541.505,A -85,B 0,C 180,E1 -28024.428,E2 -28024.428} C_VEL
LIN {X 0,Y 92.722,Z 536.411,A -85,B 0,C 180,E1 -28030.392,E2 -28030.392} C_VEL
LIN {X 0,Y 100.021,Z 529.154,A -85,B 0,C 180,E1 -28036.072,E2 -28036.072} C_VEL
LIN {X 0,Y 106.999,Z 521.114,A -85,B 0,C 180,E1 -28040.512,E2 -28040.512} C_VEL
LIN {X 0,Y 113.1,Z 512.876,A -85,B 0,C 180,E1 -28043.882,E2 -28043.882} C_VEL
LIN {X 0,Y 118.845,Z 503.819,A -85,B 0,C 180,E1 -28046.645,E2 -28046.645} C_VEL
LIN {X 0,Y 124.614,Z 493.255,A -85,B 0,C 180,E1 -28048.891,E2 -28048.891} C_VEL
LIN {X 0,Y 129.586,Z 481.707,A -85,B 0,C 180,E1 -28050.83,E2 -28050.83} C_VEL
LIN {X 0,Y 133.392,Z 470.472,A -85,B 0,C 180,E1 -28052.187,E2 -28052.187} C_VEL
LIN {X 0,Y 136.26,Z 457.97,A -85,B 0,C 180,E1 -28053.435,E2 -28053.435} C_VEL
LIN {X 0,Y 138.065,Z 445.579,A -85,B 0,C 180,E1 -28054.245,E2 -28054.245} C_VEL
LIN {X 0,Y 138.447,Z 440.758,A -85,B 0,C 180,E1 -28054.547,E2 -28054.547} C_VEL
LIN {X 0,Y 135.828,Z 434.389,A -85,B 0,C 180,E1 -28057.997,E2 -28057.997} C_VEL
LIN {X 0,Y 133.318,Z 428.947,A -85,B 0,C 180,E1 -28061.958,E2 -28061.958} C_VEL
LIN {X 0,Y 131.52,Z 425.488,A -85,B 0,C 180,E1 -28065.494,E2 -28065.494} C_VEL
LIN {X 0,Y 129.935,Z 422.1,A -85,B 0,C 180,E1 -28069.875,E2 -28069.875} C_VEL
LIN {X 0,Y 128.71,Z 418.627,A -85,B 0,C 180,E1 -28078.387,E2 -28078.387} C_VEL
LIN {X 0,Y 128.713,Z 418.915,A -85,B 0,C 180,E1 -28080.586,E2 -28080.586} C_VEL
LIN {X 0,Y 130.162,Z 422.474,A -85,B 0,C 180,E1 -28088.93,E2 -28088.93} C_VEL
LIN {X 0,Y 131.276,Z 426.431,A -85,B 0,C 180,E1 -28092.365,E2 -28092.365} C_VEL
LIN {X 0,Y 132.574,Z 431.156,A -85,B 0,C 180,E1 -28095.469,E2 -28095.469} C_VEL
LIN {X 0,Y 134.278,Z 437.561,A -85,B 0,C 180,E1 -28098.797,E2 -28098.797} C_VEL
LIN {X 0,Y 136.14,Z 445.533,A -85,B 0,C 180,E1 -28101.956,E2 -28101.956} C_VEL
LIN {X 0,Y 135.185,Z 465.995,A -85,B 0,C 180,E1 -28103.915,E2 -28103.915} C_VEL
LIN {X 0,Y 134.407,Z 471.699,A -85,B 0,C 180,E1 -28104.38,E2 -28104.38} C_VEL
LIN {X 0,Y 131.203,Z 484.799,A -85,B 0,C 180,E1 -28105.245,E2 -28105.245} C_VEL
LIN {X 0,Y 127.058,Z 496.759,A -85,B 0,C 180,E1 -28106.336,E2 -28106.336} C_VEL
LIN {X 0,Y 122.203,Z 507.87,A -85,B 0,C 180,E1 -28107.845,E2 -28107.845} C_VEL
LIN {X 0,Y 115.545,Z 519.692,A -85,B 0,C 180,E1 -28109.918,E2 -28109.918} C_VEL
LIN {X 0,Y 109.911,Z 528.287,A -85,B 0,C 180,E1 -28112.089,E2 -28112.089} C_VEL
LIN {X 0,Y 103.017,Z 537.197,A -85,B 0,C 180,E1 -28115.051,E2 -28115.051} C_VEL
LIN {X 0,Y 96.583,Z 544.603,A -85,B 0,C 180,E1 -28118.535,E2 -28118.535} C_VEL
LIN {X 0,Y 89.476,Z 551.937,A -85,B 0,C 180,E1 -28123.403,E2 -28123.403} C_VEL
LIN {X 0,Y 82.443,Z 558.615,A -85,B 0,C 180,E1 -28130.105,E2 -28130.105} C_VEL
LIN {X 0,Y 77.393,Z 563.224,A -85,B 0,C 180,E1 -28136.986,E2 -28136.986} C_VEL
LIN {X 0,Y 73.812,Z 566.711,A -85,B 0,C 180,E1 -28144.63,E2 -28144.63} C_VEL
LIN {X 0,Y 71.789,Z 569.241,A -85,B 0,C 180,E1 -28152.921,E2 -28152.921} C_VEL
LIN {X 0,Y 71.571,Z 571.186,A -85,B 0,C 180,E1 -28164.365,E2 -28164.365} C_VEL
LIN {X 0,Y 72.333,Z 571.546,A -85,B 0,C 180,E1 -28170,E2 -28170} C_VEL
LIN {X 0,Y 71.329,Z 570.638,A -85,B 0,C 180,E1 -28179.838,E2 -28179.838} C_VEL
LIN {X 0,Y 71.781,Z 569.199,A -85,B 0,C 180,E1 -28187.081,E2 -28187.081} C_VEL
LIN {X 0,Y 73.794,Z 566.641,A -85,B 0,C 180,E1 -28195.376,E2 -28195.376} C_VEL
LIN {X 0,Y 77.396,Z 563.125,A -85,B 0,C 180,E1 -28203.013,E2 -28203.013} C_VEL
LIN {X 0,Y 82.418,Z 558.501,A -85,B 0,C 180,E1 -28209.874,E2 -28209.874} C_VEL
LIN {X 0,Y 89.465,Z 551.759,A -85,B 0,C 180,E1 -28216.604,E2 -28216.604} C_VEL
LIN {X 0,Y 96.59,Z 544.383,A -85,B 0,C 180,E1 -28221.46,E2 -28221.46} C_VEL
LIN {X 0,Y 104.374,Z 535.281,A -85,B 0,C 180,E1 -28225.572,E2 -28225.572} C_VEL
LIN {X 0,Y 111.345,Z 525.988,A -85,B 0,C 180,E1 -28228.44,E2 -28228.44} C_VEL
LIN {X 0,Y 117.762,Z 515.645,A -85,B 0,C 180,E1 -28230.785,E2 -28230.785} C_VEL
LIN {X 0,Y 123.648,Z 504.209,A -85,B 0,C 180,E1 -28232.634,E2 -28232.634} C_VEL
LIN {X 0,Y 128.267,Z 492.981,A -85,B 0,C 180,E1 -28233.954,E2 -28233.954} C_VEL
LIN {X 0,Y 132.294,Z 479.997,A -85,B 0,C 180,E1 -28235.033,E2 -28235.033} C_VEL
LIN {X 0,Y 134.646,Z 468.676,A -85,B 0,C 180,E1 -28235.76,E2 -28235.76} C_VEL
LIN {X 0,Y 135.681,Z 451.909,A -85,B 0,C 180,E1 -28237.335,E2 -28237.335} C_VEL
LIN {X 0,Y 135.814,Z 445.012,A -85,B 0,C 180,E1 -28238.109,E2 -28238.109} C_VEL
LIN {X 0,Y 133.861,Z 436.643,A -85,B 0,C 180,E1 -28241.452,E2 -28241.452} C_VEL
LIN {X 0,Y 131.893,Z 429.211,A -85,B 0,C 180,E1 -28245.437,E2 -28245.437} C_VEL
LIN {X 0,Y 130.512,Z 424.444,A -85,B 0,C 180,E1 -28248.962,E2 -28248.962} C_VEL
LIN {X 0,Y 129.754,Z 421.942,A -85,B 0,C 180,E1 -28251.434,E2 -28251.434} C_VEL
LIN {X 0,Y 128.441,Z 418.094,A -85,B 0,C 180,E1 -28260,E2 -28260} C_VEL
LIN {X 0,Y 128.432,Z 418.253,A -85,B 0,C 180,E1 -28262.25,E2 -28262.25} C_VEL
LIN {X 0,Y 128.478,Z 419.909,A -85,B 0,C 180,E1 -28264.783,E2 -28264.783} C_VEL
LIN {X 0,Y 128.625,Z 422.499,A -85,B 0,C 180,E1 -28267.168,E2 -28267.168} C_VEL
LIN {X 0,Y 129.343,Z 428.884,A -85,B 0,C 180,E1 -28271.696,E2 -28271.696} C_VEL
LIN {X 0,Y 130.353,Z 432.826,A -85,B 0,C 180,E1 -28274.762,E2 -28274.762} C_VEL
LIN {X 0,Y 132.271,Z 437.103,A -85,B 0,C 180,E1 -28278.591,E2 -28278.591} C_VEL
LIN {X 0,Y 134.491,Z 442.524,A -85,B 0,C 180,E1 -28282.163,E2 -28282.163} C_VEL
LIN {X 0,Y 135.085,Z 444.121,A -85,B 0,C 180,E1 -28283.031,E2 -28283.031} C_VEL
LIN {X 0,Y 133.193,Z 457.771,A -85,B 0,C 180,E1 -28283.908,E2 -28283.908} C_VEL
LIN {X 0,Y 130.172,Z 470.451,A -85,B 0,C 180,E1 -28285.023,E2 -28285.023} C_VEL
LIN {X 0,Y 126.209,Z 482.21,A -85,B 0,C 180,E1 -28286.455,E2 -28286.455} C_VEL
LIN {X 0,Y 121.171,Z 493.531,A -85,B 0,C 180,E1 -28288.249,E2 -28288.249} C_VEL
LIN {X 0,Y 115.183,Z 504.264,A -85,B 0,C 180,E1 -28290.477,E2 -28290.477} C_VEL
LIN {X 0,Y 109.112,Z 513.436,A -85,B 0,C 180,E1 -28293.142,E2 -28293.142} C_VEL
LIN {X 0,Y 102.684,Z 521.762,A -85,B 0,C 180,E1 -28296.468,E2 -28296.468} C_VEL
LIN {X 0,Y 95.272,Z 529.862,A -85,B 0,C 180,E1 -28300.878,E2 -28300.878} C_VEL
LIN {X 0,Y 87.744,Z 536.959,A -85,B 0,C 180,E1 -28306.447,E2 -28306.447} C_VEL
LIN {X 0,Y 81.334,Z 542.319,A -85,B 0,C 180,E1 -28312.782,E2 -28312.782} C_VEL
LIN {X 0,Y 75.988,Z 546.201,A -85,B 0,C 180,E1 -28319.424,E2 -28319.424} C_VEL
LIN {X 0,Y 71.533,Z 549.086,A -85,B 0,C 180,E1 -28326.86,E2 -28326.86} C_VEL
LIN {X 0,Y 69.612,Z 550.411,A -85,B 0,C 180,E1 -28332.37,E2 -28332.37} C_VEL
LIN {X 0,Y 67.22,Z 551.95,A -85,B 0,C 180,E1 -28343.999,E2 -28343.999} C_VEL
LIN {X 0,Y 66.913,Z 552.169,A -85,B 0,C 180,E1 -28350,E2 -28350} C_VEL
LIN {X 0,Y 67.219,Z 551.976,A -85,B 0,C 180,E1 -28356.001,E2 -28356.001} C_VEL
LIN {X 0,Y 69.603,Z 550.47,A -85,B 0,C 180,E1 -28367.633,E2 -28367.633} C_VEL
LIN {X 0,Y 71.514,Z 549.174,A -85,B 0,C 180,E1 -28373.147,E2 -28373.147} C_VEL
LIN {X 0,Y 75.981,Z 546.32,A -85,B 0,C 180,E1 -28380.579,E2 -28380.579} C_VEL
LIN {X 0,Y 81.314,Z 542.482,A -85,B 0,C 180,E1 -28387.229,E2 -28387.229} C_VEL
LIN {X 0,Y 87.488,Z 537.387,A -85,B 0,C 180,E1 -28393.376,E2 -28393.376} C_VEL
LIN {X 0,Y 95.279,Z 530.13,A -85,B 0,C 180,E1 -28399.117,E2 -28399.117} C_VEL
LIN {X 0,Y 102.672,Z 522.089,A -85,B 0,C 180,E1 -28403.541,E2 -28403.541} C_VEL
LIN {X 0,Y 109.104,Z 513.852,A -85,B 0,C 180,E1 -28406.866,E2 -28406.866} C_VEL
LIN {X 0,Y 115.129,Z 504.793,A -85,B 0,C 180,E1 -28409.569,E2 -28409.569} C_VEL
LIN {X 0,Y 121.134,Z 494.227,A -85,B 0,C 180,E1 -28411.738,E2 -28411.738} C_VEL
LIN {X 0,Y 126.345,Z 482.6,A -85,B 0,C 180,E1 -28413.623,E2 -28413.623} C_VEL
LIN {X 0,Y 130.48,Z 470.702,A -85,B 0,C 180,E1 -28415,E2 -28415} C_VEL
LIN {X 0,Y 133.48,Z 457.773,A -85,B 0,C 180,E1 -28416.231,E2 -28416.231} C_VEL
LIN {X 0,Y 135.357,Z 444.373,A -85,B 0,C 180,E1 -28417.08,E2 -28417.08} C_VEL
LIN {X 0,Y 133.01,Z 438.466,A -85,B 0,C 180,E1 -28420.72,E2 -28420.72} C_VEL
LIN {X 0,Y 131.316,Z 434.568,A -85,B 0,C 180,E1 -28423.881,E2 -28423.881} C_VEL
LIN {X 0,Y 130.055,Z 431.878,A -85,B 0,C 180,E1 -28426.754,E2 -28426.754} C_VEL
LIN {X 0,Y 128.834,Z 428.975,A -85,B 0,C 180,E1 -28430.581,E2 -28430.581} C_VEL
LIN {X 0,Y 127.832,Z 425.776,A -85,B 0,C 180,E1 -28438.376,E2 -28438.376} C_VEL
LIN {X 0,Y 127.831,Z 426.095,A -85,B 0,C 180,E1 -28440.59,E2 -28440.59} C_VEL
LIN {X 0,Y 128.98,Z 429.245,A -85,B 0,C 180,E1 -28448.026,E2 -28448.026} C_VEL
LIN {X 0,Y 129.798,Z 432.715,A -85,B 0,C 180,E1 -28451.023,E2 -28451.023} C_VEL
LIN {X 0,Y 130.89,Z 437.312,A -85,B 0,C 180,E1 -28454.081,E2 -28454.081} C_VEL
LIN {X 0,Y 132.381,Z 443.956,A -85,B 0,C 180,E1 -28457.474,E2 -28457.474} C_VEL
LIN {X 0,Y 133.349,Z 449.024,A -85,B 0,C 180,E1 -28459.463,E2 -28459.463} C_VEL
LIN {X 0,Y 132.161,Z 466.81,A -85,B 0,C 180,E1 -28461.177,E2 -28461.177} C_VEL
LIN {X 0,Y 131.382,Z 471.872,A -85,B 0,C 180,E1 -28461.612,E2 -28461.612} C_VEL
LIN {X 0,Y 128.185,Z 484.305,A -85,B 0,C 180,E1 -28462.407,E2 -28462.407} C_VEL
LIN {X 0,Y 123.79,Z 496.459,A -85,B 0,C 180,E1 -28463.466,E2 -28463.466} C_VEL
LIN {X 0,Y 118.283,Z 508.321,A -85,B 0,C 180,E1 -28465.029,E2 -28465.029} C_VEL
LIN {X 0,Y 111.417,Z 519.89,A -85,B 0,C 180,E1 -28467.005,E2 -28467.005} C_VEL
LIN {X 0,Y 104.847,Z 529.261,A -85,B 0,C 180,E1 -28469.379,E2 -28469.379} C_VEL
LIN {X 0,Y 96.336,Z 539.322,A -85,B 0,C 180,E1 -28472.971,E2 -28472.971} C_VEL
LIN {X 0,Y 88.449,Z 547.479,A -85,B 0,C 180,E1 -28477.385,E2 -28477.385} C_VEL
LIN {X 0,Y 81.262,Z 554.064,A -85,B 0,C 180,E1 -28482.683,E2 -28482.683} C_VEL
LIN {X 0,Y 75.038,Z 559.356,A -85,B 0,C 180,E1 -28489.035,E2 -28489.035} C_VEL
LIN {X 0,Y 69.96,Z 563.522,A -85,B 0,C 180,E1 -28496.461,E2 -28496.461} C_VEL
LIN {X 0,Y 66.411,Z 566.686,A -85,B 0,C 180,E1 -28504.957,E2 -28504.957} C_VEL
LIN {X 0,Y 64.318,Z 569.41,A -85,B 0,C 180,E1 -28517.377,E2 -28517.377} C_VEL
LIN {X 0,Y 64.445,Z 570.189,A -85,B 0,C 180,E1 -28523.739,E2 -28523.739} C_VEL
LIN {X 0,Y 65.218,Z 570.555,A -85,B 0,C 180,E1 -28530,E2 -28530} C_VEL
LIN {X 0,Y 64.279,Z 569.743,A -85,B 0,C 180,E1 -28540.257,E2 -28540.257} C_VEL
LIN {X 0,Y 64.969,Z 568.202,A -85,B 0,C 180,E1 -28548.936,E2 -28548.936} C_VEL
LIN {X 0,Y 67.391,Z 565.643,A -85,B 0,C 180,E1 -28557.988,E2 -28557.988} C_VEL
LIN {X 0,Y 71.488,Z 562.126,A -85,B 0,C 180,E1 -28566.146,E2 -28566.146} C_VEL
LIN {X 0,Y 77.322,Z 557.288,A -85,B 0,C 180,E1 -28573.565,E2 -28573.565} C_VEL
LIN {X 0,Y 84.708,Z 550.761,A -85,B 0,C 180,E1 -28580.124,E2 -28580.124} C_VEL
LIN {X 0,Y 92.299,Z 543.384,A -85,B 0,C 180,E1 -28584.938,E2 -28584.938} C_VEL
LIN {X 0,Y 100.532,Z 534.292,A -85,B 0,C 180,E1 -28588.91,E2 -28588.91} C_VEL
LIN {X 0,Y 107.807,Z 524.999,A -85,B 0,C 180,E1 -28591.649,E2 -28591.649} C_VEL
LIN {X 0,Y 114.465,Z 514.653,A -85,B 0,C 180,E1 -28593.888,E2 -28593.888} C_VEL
LIN {X 0,Y 120.536,Z 503.212,A -85,B 0,C 180,E1 -28595.646,E2 -28595.646} C_VEL
LIN {X 0,Y 125.511,Z 491.431,A -85,B 0,C 180,E1 -28596.94,E2 -28596.94} C_VEL
LIN {X 0,Y 129.526,Z 478.683,A -85,B 0,C 180,E1 -28597.913,E2 -28597.913} C_VEL
LIN {X 0,Y 131.63,Z 468.995,A -85,B 0,C 180,E1 -28598.551,E2 -28598.551} C_VEL
LIN {X 0,Y 132.872,Z 453.454,A -85,B 0,C 180,E1 -28600.041,E2 -28600.041} C_VEL
LIN {X 0,Y 133.04,Z 448.253,A -85,B 0,C 180,E1 -28600.629,E2 -28600.629} C_VEL
LIN {X 0,Y 131.498,Z 440.92,A -85,B 0,C 180,E1 -28603.804,E2 -28603.804} C_VEL
LIN {X 0,Y 130.07,Z 434.669,A -85,B 0,C 180,E1 -28607.332,E2 -28607.332} C_VEL
LIN {X 0,Y 129.06,Z 430.504,A -85,B 0,C 180,E1 -28610.499,E2 -28610.499} C_VEL
LIN {X 0,Y 128.64,Z 428.789,A -85,B 0,C 180,E1 -28612.15,E2 -28612.15} C_VEL
LIN {X 0,Y 127.552,Z 425.328,A -85,B 0,C 180,E1 -28620,E2 -28620} C_VEL
LIN {X 0,Y 127.554,Z 425.309,A -85,B 0,C 180,E1 -28621.974,E2 -28621.974} C_VEL
LIN {X 0,Y 128.839,Z 429.411,A -85,B 0,C 180,E1 -28630.61,E2 -28630.61} C_VEL
LIN {X 0,Y 130.353,Z 432.826,A -85,B 0,C 180,E1 -28634.762,E2 -28634.762} C_VEL
LIN {X 0,Y 131.224,Z 435.779,A -85,B 0,C 180,E1 -28636.811,E2 -28636.811} C_VEL
LIN {X 0,Y 131.918,Z 439.685,A -85,B 0,C 180,E1 -28638.535,E2 -28638.535} C_VEL
LIN {X 0,Y 132.27,Z 444.31,A -85,B 0,C 180,E1 -28639.816,E2 -28639.816} C_VEL
LIN {X 0,Y 132.093,Z 448.849,A -85,B 0,C 180,E1 -28640.451,E2 -28640.451} C_VEL
LIN {X 0,Y 132.02,Z 449.522,A -85,B 0,C 180,E1 -28640.493,E2 -28640.493} C_VEL
LIN {X 0,Y 129.765,Z 462.265,A -85,B 0,C 180,E1 -28641.34,E2 -28641.34} C_VEL
LIN {X 0,Y 126.49,Z 474.188,A -85,B 0,C 180,E1 -28642.451,E2 -28642.451} C_VEL
LIN {X 0,Y 122.053,Z 486.011,A -85,B 0,C 180,E1 -28643.917,E2 -28643.917} C_VEL
LIN {X 0,Y 116.873,Z 496.638,A -85,B 0,C 180,E1 -28645.579,E2 -28645.579} C_VEL
LIN {X 0,Y 111.02,Z 506.399,A -85,B 0,C 180,E1 -28647.596,E2 -28647.596} C_VEL
LIN {X 0,Y 104.052,Z 516.192,A -85,B 0,C 180,E1 -28650.553,E2 -28650.553} C_VEL
LIN {X 0,Y 95.971,Z 525.657,A -85,B 0,C 180,E1 -28654.53,E2 -28654.53} C_VEL
LIN {X 0,Y 88.19,Z 533.302,A -85,B 0,C 180,E1 -28659.197,E2 -28659.197} C_VEL
LIN {X 0,Y 80.103,Z 540.096,A -85,B 0,C 180,E1 -28665.421,E2 -28665.421} C_VEL
LIN {X 0,Y 73.772,Z 544.698,A -85,B 0,C 180,E1 -28671.741,E2 -28671.741} C_VEL
LIN {X 0,Y 68.166,Z 548.245,A -85,B 0,C 180,E1 -28678.97,E2 -28678.97} C_VEL
LIN {X 0,Y 65.126,Z 550.066,A -85,B 0,C 180,E1 -28684.428,E2 -28684.428} C_VEL
LIN {X 0,Y 62.948,Z 551.389,A -85,B 0,C 180,E1 -28690.431,E2 -28690.431} C_VEL
LIN {X 0,Y 60.235,Z 552.928,A -85,B 0,C 180,E1 -28703.3,E2 -28703.3} C_VEL
LIN {X 0,Y 59.885,Z 553.147,A -85,B 0,C 180,E1 -28710,E2 -28710} C_VEL
LIN {X 0,Y 60.234,Z 552.954,A -85,B 0,C 180,E1 -28716.7,E2 -28716.7} C_VEL
LIN {X 0,Y 62.939,Z 551.448,A -85,B 0,C 180,E1 -28729.572,E2 -28729.572} C_VEL
LIN {X 0,Y 65.107,Z 550.152,A -85,B 0,C 180,E1 -28735.58,E2 -28735.58} C_VEL
LIN {X 0,Y 70.022,Z 547.297,A -85,B 0,C 180,E1 -28743.506,E2 -28743.506} C_VEL
LIN {X 0,Y 75.837,Z 543.458,A -85,B 0,C 180,E1 -28750.443,E2 -28750.443} C_VEL
LIN {X 0,Y 82.521,Z 538.363,A -85,B 0,C 180,E1 -28756.73,E2 -28756.73} C_VEL
LIN {X 0,Y 90.835,Z 531.106,A -85,B 0,C 180,E1 -28762.471,E2 -28762.471} C_VEL
LIN {X 0,Y 98.658,Z 523.065,A -85,B 0,C 180,E1 -28766.826,E2 -28766.826} C_VEL
LIN {X 0,Y 105.425,Z 514.827,A -85,B 0,C 180,E1 -28770.067,E2 -28770.067} C_VEL
LIN {X 0,Y 111.729,Z 505.769,A -85,B 0,C 180,E1 -28772.682,E2 -28772.682} C_VEL
LIN {X 0,Y 117.969,Z 495.2,A -85,B 0,C 180,E1 -28774.744,E2 -28774.744} C_VEL
LIN {X 0,Y 123.296,Z 483.788,A -85,B 0,C 180,E1 -28776.514,E2 -28776.514} C_VEL
LIN {X 0,Y 127.75,Z 471.373,A -85,B 0,C 180,E1 -28777.892,E2 -28777.892} C_VEL
LIN {X 0,Y 130.87,Z 458.409,A -85,B 0,C 180,E1 -28779.074,E2 -28779.074} C_VEL
LIN {X 0,Y 132.447,Z 448,A -85,B 0,C 180,E1 -28779.773,E2 -28779.773} C_VEL
LIN {X 0,Y 130.225,Z 441.887,A -85,B 0,C 180,E1 -28784.144,E2 -28784.144} C_VEL
LIN {X 0,Y 128.712,Z 438.431,A -85,B 0,C 180,E1 -28787.867,E2 -28787.867} C_VEL
LIN {X 0,Y 127.729,Z 435.805,A -85,B 0,C 180,E1 -28791.396,E2 -28791.396} C_VEL
LIN {X 0,Y 126.96,Z 432.889,A -85,B 0,C 180,E1 -28798.364,E2 -28798.364} C_VEL
LIN {X 0,Y 126.948,Z 433.287,A -85,B 0,C 180,E1 -28800.595,E2 -28800.595} C_VEL
LIN {X 0,Y 127.82,Z 435.969,A -85,B 0,C 180,E1 -28807.057,E2 -28807.057} C_VEL
LIN {X 0,Y 128.423,Z 439.091,A -85,B 0,C 180,E1 -28809.746,E2 -28809.746} C_VEL
LIN {X 0,Y 129.345,Z 443.837,A -85,B 0,C 180,E1 -28812.852,E2 -28812.852} C_VEL
LIN {X 0,Y 130.574,Z 450.571,A -85,B 0,C 180,E1 -28816.177,E2 -28816.177} C_VEL
LIN {X 0,Y 130.826,Z 452.139,A -85,B 0,C 180,E1 -28816.81,E2 -28816.81} C_VEL
LIN {X 0,Y 129.477,Z 467.485,A -85,B 0,C 180,E1 -28818.313,E2 -28818.313} C_VEL
LIN {X 0,Y 128.41,Z 473.359,A -85,B 0,C 180,E1 -28818.804,E2 -28818.804} C_VEL
LIN {X 0,Y 124.769,Z 485.984,A -85,B 0,C 180,E1 -28819.597,E2 -28819.597} C_VEL
LIN {X 0,Y 120.138,Z 497.715,A -85,B 0,C 180,E1 -28820.614,E2 -28820.614} C_VEL
LIN {X 0,Y 114.651,Z 508.801,A -85,B 0,C 180,E1 -28822.032,E2 -28822.032} C_VEL
LIN {X 0,Y 107.6,Z 520.037,A -85,B 0,C 180,E1 -28823.878,E2 -28823.878} C_VEL
LIN {X 0,Y 101.555,Z 528.277,A -85,B 0,C 180,E1 -28825.89,E2 -28825.89} C_VEL
LIN {X 0,Y 92.655,Z 538.334,A -85,B 0,C 180,E1 -28829.276,E2 -28829.276} C_VEL
LIN {X 0,Y 84.299,Z 546.486,A -85,B 0,C 180,E1 -28833.52,E2 -28833.52} C_VEL
LIN {X 0,Y 76.581,Z 553.068,A -85,B 0,C 180,E1 -28838.735,E2 -28838.735} C_VEL
LIN {X 0,Y 69.794,Z 558.362,A -85,B 0,C 180,E1 -28845.181,E2 -28845.181} C_VEL
LIN {X 0,Y 64.107,Z 562.526,A -85,B 0,C 180,E1 -28852.918,E2 -28852.918} C_VEL
LIN {X 0,Y 59.997,Z 565.69,A -85,B 0,C 180,E1 -28862.06,E2 -28862.06} C_VEL
LIN {X 0,Y 57.342,Z 568.412,A -85,B 0,C 180,E1 -28875.811,E2 -28875.811} C_VEL
LIN {X 0,Y 57.33,Z 569.192,A -85,B 0,C 180,E1 -28882.959,E2 -28882.959} C_VEL
LIN {X 0,Y 58.1,Z 569.565,A -85,B 0,C 180,E1 -28890,E2 -28890} C_VEL
LIN {X 0,Y 57.244,Z 568.825,A -85,B 0,C 180,E1 -28900.831,E2 -28900.831} C_VEL
LIN {X 0,Y 58.23,Z 567.203,A -85,B 0,C 180,E1 -28911.228,E2 -28911.228} C_VEL
LIN {X 0,Y 61.145,Z 564.643,A -85,B 0,C 180,E1 -28921.146,E2 -28921.146} C_VEL
LIN {X 0,Y 65.84,Z 561.128,A -85,B 0,C 180,E1 -28929.826,E2 -28929.826} C_VEL
LIN {X 0,Y 72.029,Z 556.502,A -85,B 0,C 180,E1 -28937.199,E2 -28937.199} C_VEL
LIN {X 0,Y 80.319,Z 549.766,A -85,B 0,C 180,E1 -28944.034,E2 -28944.034} C_VEL
LIN {X 0,Y 88.39,Z 542.388,A -85,B 0,C 180,E1 -28948.73,E2 -28948.73} C_VEL
LIN {X 0,Y 97.059,Z 533.302,A -85,B 0,C 180,E1 -28952.499,E2 -28952.499} C_VEL
LIN {X 0,Y 104.631,Z 524.011,A -85,B 0,C 180,E1 -28955.063,E2 -28955.063} C_VEL
LIN {X 0,Y 110.74,Z 514.949,A -85,B 0,C 180,E1 -28956.957,E2 -28956.957} C_VEL
LIN {X 0,Y 116.997,Z 503.812,A -85,B 0,C 180,E1 -28958.602,E2 -28958.602} C_VEL
LIN {X 0,Y 122.533,Z 491.356,A -85,B 0,C 180,E1 -28959.911,E2 -28959.911} C_VEL
LIN {X 0,Y 126.53,Z 479.525,A -85,B 0,C 180,E1 -28960.775,E2 -28960.775} C_VEL
LIN {X 0,Y 128.837,Z 469.732,A -85,B 0,C 180,E1 -28961.399,E2 -28961.399} C_VEL
LIN {X 0,Y 130.304,Z 456.196,A -85,B 0,C 180,E1 -28962.742,E2 -28962.742} C_VEL
LIN {X 0,Y 130.506,Z 451.587,A -85,B 0,C 180,E1 -28963.274,E2 -28963.274} C_VEL
LIN {X 0,Y 129.338,Z 444.998,A -85,B 0,C 180,E1 -28966.325,E2 -28966.325} C_VEL
LIN {X 0,Y 128.431,Z 440.288,A -85,B 0,C 180,E1 -28969.158,E2 -28969.158} C_VEL
LIN {X 0,Y 127.744,Z 436.771,A -85,B 0,C 180,E1 -28971.878,E2 -28971.878} C_VEL
LIN {X 0,Y 127.436,Z 435.457,A -85,B 0,C 180,E1 -28973.309,E2 -28973.309} C_VEL
LIN {X 0,Y 126.668,Z 432.532,A -85,B 0,C 180,E1 -28980,E2 -28980} C_VEL
LIN {X 0,Y 126.665,Z 432.588,A -85,B 0,C 180,E1 -28982.107,E2 -28982.107} C_VEL
LIN {X 0,Y 127.667,Z 436.108,A -85,B 0,C 180,E1 -28989.669,E2 -28989.669} C_VEL
LIN {X 0,Y 129.147,Z 439.86,A -85,B 0,C 180,E1 -28994.175,E2 -28994.175} C_VEL
LIN {X 0,Y 130.87,Z 444.091,A -85,B 0,C 180,E1 -28997.885,E2 -28997.885} C_VEL
LIN {X 0,Y 132.164,Z 447.733,A -85,B 0,C 180,E1 -29000.324,E2 -29000.324} C_VEL
LIN {X 0,Y 132.02,Z 449.522,A -85,B 0,C 180,E1 -29000.493,E2 -29000.493} C_VEL
LIN {X 0,Y 130.991,Z 455.345,A -85,B 0,C 180,E1 -29000.552,E2 -29000.552} C_VEL
LIN {X 0,Y 128.178,Z 464.786,A -85,B 0,C 180,E1 -29000.035,E2 -29000.035} C_VEL
LIN {X 0,Y 124.651,Z 473.994,A -85,B 0,C 180,E1 -28999.64,E2 -28999.64} C_VEL
LIN {X 0,Y 122.488,Z 479.445,A -85,B 0,C 180,E1 -28999.929,E2 -28999.929} C_VEL
LIN {X 0,Y 117.502,Z 491.032,A -85,B 0,C 180,E1 -29001.429,E2 -29001.429} C_VEL
LIN {X 0,Y 111.76,Z 501.481,A -85,B 0,C 180,E1 -29003.121,E2 -29003.121} C_VEL
LIN {X 0,Y 106.477,Z 509.481,A -85,B 0,C 180,E1 -29004.831,E2 -29004.831} C_VEL
LIN {X 0,Y 99.239,Z 518.912,A -85,B 0,C 180,E1 -29007.722,E2 -29007.722} C_VEL
LIN {X 0,Y 92.169,Z 526.638,A -85,B 0,C 180,E1 -29010.929,E2 -29010.929} C_VEL
LIN {X 0,Y 83.926,Z 534.281,A -85,B 0,C 180,E1 -29015.476,E2 -29015.476} C_VEL
LIN {X 0,Y 75.258,Z 541.075,A -85,B 0,C 180,E1 -29021.663,E2 -29021.663} C_VEL
LIN {X 0,Y 68.392,Z 545.677,A -85,B 0,C 180,E1 -29028.093,E2 -29028.093} C_VEL
LIN {X 0,Y 62.247,Z 549.224,A -85,B 0,C 180,E1 -29035.631,E2 -29035.631} C_VEL
LIN {X 0,Y 58.861,Z 551.045,A -85,B 0,C 180,E1 -29041.472,E2 -29041.472} C_VEL
LIN {X 0,Y 56.373,Z 552.368,A -85,B 0,C 180,E1 -29048.038,E2 -29048.038} C_VEL
LIN {X 0,Y 53.261,Z 553.906,A -85,B 0,C 180,E1 -29062.418,E2 -29062.418} C_VEL
LIN {X 0,Y 52.857,Z 554.125,A -85,B 0,C 180,E1 -29070,E2 -29070} C_VEL
LIN {X 0,Y 53.26,Z 553.932,A -85,B 0,C 180,E1 -29077.583,E2 -29077.583} C_VEL
LIN {X 0,Y 56.364,Z 552.426,A -85,B 0,C 180,E1 -29091.966,E2 -29091.966} C_VEL
LIN {X 0,Y 58.843,Z 551.13,A -85,B 0,C 180,E1 -29098.538,E2 -29098.538} C_VEL
LIN {X 0,Y 64.279,Z 548.275,A -85,B 0,C 180,E1 -29106.966,E2 -29106.966} C_VEL
LIN {X 0,Y 70.636,Z 544.435,A -85,B 0,C 180,E1 -29114.144,E2 -29114.144} C_VEL
LIN {X 0,Y 77.872,Z 539.34,A -85,B 0,C 180,E1 -29120.497,E2 -29120.497} C_VEL
LIN {X 0,Y 86.733,Z 532.082,A -85,B 0,C 180,E1 -29126.155,E2 -29126.155} C_VEL
LIN {X 0,Y 94.994,Z 524.041,A -85,B 0,C 180,E1 -29130.377,E2 -29130.377} C_VEL
LIN {X 0,Y 102.099,Z 515.802,A -85,B 0,C 180,E1 -29133.488,E2 -29133.488} C_VEL
LIN {X 0,Y 108.681,Z 506.744,A -85,B 0,C 180,E1 -29135.979,E2 -29135.979} C_VEL
LIN {X 0,Y 115.144,Z 496.176,A -85,B 0,C 180,E1 -29137.91,E2 -29137.91} C_VEL
LIN {X 0,Y 120.632,Z 484.836,A -85,B 0,C 180,E1 -29139.57,E2 -29139.57} C_VEL
LIN {X 0,Y 124.928,Z 473.449,A -85,B 0,C 180,E1 -29140.769,E2 -29140.769} C_VEL
LIN {X 0,Y 128.299,Z 460.502,A -85,B 0,C 180,E1 -29141.92,E2 -29141.92} C_VEL
LIN {X 0,Y 129.809,Z 451.937,A -85,B 0,C 180,E1 -29142.513,E2 -29142.513} C_VEL
LIN {X 0,Y 128.461,Z 447.67,A -85,B 0,C 180,E1 -29145.95,E2 -29145.95} C_VEL
LIN {X 0,Y 127.347,Z 444.734,A -85,B 0,C 180,E1 -29149.265,E2 -29149.265} C_VEL
LIN {X 0,Y 126.696,Z 442.691,A -85,B 0,C 180,E1 -29152.028,E2 -29152.028} C_VEL
LIN {X 0,Y 126.078,Z 440.071,A -85,B 0,C 180,E1 -29158.353,E2 -29158.353} C_VEL
LIN {X 0,Y 126.072,Z 440.584,A -85,B 0,C 180,E1 -29160.898,E2 -29160.898} C_VEL
LIN {X 0,Y 126.715,Z 442.777,A -85,B 0,C 180,E1 -29166.169,E2 -29166.169} C_VEL
LIN {X 0,Y 127.191,Z 446.04,A -85,B 0,C 180,E1 -29168.84,E2 -29168.84} C_VEL
LIN {X 0,Y 127.961,Z 451.136,A -85,B 0,C 180,E1 -29171.986,E2 -29171.986} C_VEL
LIN {X 0,Y 128.566,Z 455.394,A -85,B 0,C 180,E1 -29174.04,E2 -29174.04} C_VEL
LIN {X 0,Y 127.051,Z 468.318,A -85,B 0,C 180,E1 -29175.36,E2 -29175.36} C_VEL
LIN {X 0,Y 125.805,Z 474.243,A -85,B 0,C 180,E1 -29175.828,E2 -29175.828} C_VEL
LIN {X 0,Y 121.599,Z 487.698,A -85,B 0,C 180,E1 -29176.654,E2 -29176.654} C_VEL
LIN {X 0,Y 116.254,Z 500.093,A -85,B 0,C 180,E1 -29177.717,E2 -29177.717} C_VEL
LIN {X 0,Y 109.78,Z 511.827,A -85,B 0,C 180,E1 -29179.22,E2 -29179.22} C_VEL
LIN {X 0,Y 102.543,Z 522.293,A -85,B 0,C 180,E1 -29180.965,E2 -29180.965} C_VEL
LIN {X 0,Y 95.523,Z 530.899,A -85,B 0,C 180,E1 -29183.123,E2 -29183.123} C_VEL
LIN {X 0,Y 86.376,Z 540.245,A -85,B 0,C 180,E1 -29186.491,E2 -29186.491} C_VEL
LIN {X 0,Y 77.744,Z 547.82,A -85,B 0,C 180,E1 -29190.82,E2 -29190.82} C_VEL
LIN {X 0,Y 69.753,Z 553.956,A -85,B 0,C 180,E1 -29196.29,E2 -29196.29} C_VEL
LIN {X 0,Y 62.665,Z 558.866,A -85,B 0,C 180,E1 -29203.2,E2 -29203.2} C_VEL
LIN {X 0,Y 56.764,Z 562.677,A -85,B 0,C 180,E1 -29211.754,E2 -29211.754} C_VEL
LIN {X 0,Y 53.757,Z 564.691,A -85,B 0,C 180,E1 -29218.471,E2 -29218.471} C_VEL
LIN {X 0,Y 50.434,Z 567.417,A -85,B 0,C 180,E1 -29233.817,E2 -29233.817} C_VEL
LIN {X 0,Y 50.233,Z 568.196,A -85,B 0,C 180,E1 -29241.957,E2 -29241.957} C_VEL
LIN {X 0,Y 50.98,Z 568.574,A -85,B 0,C 180,E1 -29250,E2 -29250} C_VEL
LIN {X 0,Y 50.431,Z 567.385,A -85,B 0,C 180,E1 -29266.183,E2 -29266.183} C_VEL
LIN {X 0,Y 53.747,Z 564.624,A -85,B 0,C 180,E1 -29281.536,E2 -29281.536} C_VEL
LIN {X 0,Y 58.556,Z 561.439,A -85,B 0,C 180,E1 -29291.308,E2 -29291.308} C_VEL
LIN {X 0,Y 65.578,Z 556.763,A -85,B 0,C 180,E1 -29299.983,E2 -29299.983} C_VEL
LIN {X 0,Y 73.632,Z 550.874,A -85,B 0,C 180,E1 -29306.631,E2 -29306.631} C_VEL
LIN {X 0,Y 82.012,Z 544.022,A -85,B 0,C 180,E1 -29311.445,E2 -29311.445} C_VEL
LIN {X 0,Y 90.898,Z 535.575,A -85,B 0,C 180,E1 -29315.293,E2 -29315.293} C_VEL
LIN {X 0,Y 98.666,Z 526.963,A -85,B 0,C 180,E1 -29317.816,E2 -29317.816} C_VEL
LIN {X 0,Y 106.548,Z 516.332,A -85,B 0,C 180,E1 -29320.039,E2 -29320.039} C_VEL
LIN {X 0,Y 112.909,Z 505.965,A -85,B 0,C 180,E1 -29321.539,E2 -29321.539} C_VEL
LIN {X 0,Y 118.838,Z 493.895,A -85,B 0,C 180,E1 -29322.801,E2 -29322.801} C_VEL
LIN {X 0,Y 123.484,Z 481.354,A -85,B 0,C 180,E1 -29323.705,E2 -29323.705} C_VEL
LIN {X 0,Y 126.428,Z 470.112,A -85,B 0,C 180,E1 -29324.407,E2 -29324.407} C_VEL
LIN {X 0,Y 128.246,Z 455.929,A -85,B 0,C 180,E1 -29325.823,E2 -29325.823} C_VEL
LIN {X 0,Y 128.233,Z 454.638,A -85,B 0,C 180,E1 -29326.125,E2 -29326.125} C_VEL
LIN {X 0,Y 127.205,Z 447.539,A -85,B 0,C 180,E1 -29329.857,E2 -29329.857} C_VEL
LIN {X 0,Y 126.539,Z 443.18,A -85,B 0,C 180,E1 -29333.113,E2 -29333.113} C_VEL
LIN {X 0,Y 126.304,Z 442.139,A -85,B 0,C 180,E1 -29334.412,E2 -29334.412} C_VEL
LIN {X 0,Y 125.785,Z 439.722,A -85,B 0,C 180,E1 -29340,E2 -29340} C_VEL
LIN {X 0,Y 125.781,Z 439.795,A -85,B 0,C 180,E1 -29342.122,E2 -29342.122} C_VEL
LIN {X 0,Y 126.591,Z 442.988,A -85,B 0,C 180,E1 -29348.983,E2 -29348.983} C_VEL
LIN {X 0,Y 127.857,Z 446.615,A -85,B 0,C 180,E1 -29353.308,E2 -29353.308} C_VEL
LIN {X 0,Y 129.155,Z 450.458,A -85,B 0,C 180,E1 -29356.681,E2 -29356.681} C_VEL
LIN {X 0,Y 129.544,Z 451.732,A -85,B 0,C 180,E1 -29357.615,E2 -29357.615} C_VEL
LIN {X 0,Y 126.926,Z 465.026,A -85,B 0,C 180,E1 -29358.522,E2 -29358.522} C_VEL
LIN {X 0,Y 123.146,Z 477.647,A -85,B 0,C 180,E1 -29359.717,E2 -29359.717} C_VEL
LIN {X 0,Y 122.488,Z 479.445,A -85,B 0,C 180,E1 -29359.929,E2 -29359.929} C_VEL
LIN {X 0,Y 120.126,Z 484.902,A -85,B 0,C 180,E1 -29360.287,E2 -29360.287} C_VEL
LIN {X 0,Y 115.309,Z 493.535,A -85,B 0,C 180,E1 -29360.177,E2 -29360.177} C_VEL
LIN {X 0,Y 109.864,Z 501.765,A -85,B 0,C 180,E1 -29360.067,E2 -29360.067} C_VEL
LIN {X 0,Y 106.527,Z 506.52,A -85,B 0,C 180,E1 -29360.484,E2 -29360.484} C_VEL
LIN {X 0,Y 99.168,Z 516.38,A -85,B 0,C 180,E1 -29362.884,E2 -29362.884} C_VEL
LIN {X 0,Y 91.732,Z 524.703,A -85,B 0,C 180,E1 -29365.816,E2 -29365.816} C_VEL
LIN {X 0,Y 83.019,Z 532.802,A -85,B 0,C 180,E1 -29369.807,E2 -29369.807} C_VEL
LIN {X 0,Y 73.906,Z 539.898,A -85,B 0,C 180,E1 -29375.111,E2 -29375.111} C_VEL
LIN {X 0,Y 65.792,Z 545.257,A -85,B 0,C 180,E1 -29381.605,E2 -29381.605} C_VEL
LIN {X 0,Y 58.821,Z 549.138,A -85,B 0,C 180,E1 -29388.919,E2 -29388.919} C_VEL
LIN {X 0,Y 52.79,Z 552.024,A -85,B 0,C 180,E1 -29397.825,E2 -29397.825} C_VEL
LIN {X 0,Y 49.923,Z 553.347,A -85,B 0,C 180,E1 -29405.019,E2 -29405.019} C_VEL
LIN {X 0,Y 46.303,Z 554.884,A -85,B 0,C 180,E1 -29421.27,E2 -29421.27} C_VEL
LIN {X 0,Y 45.829,Z 555.103,A -85,B 0,C 180,E1 -29430,E2 -29430} C_VEL
LIN {X 0,Y 46.303,Z 554.909,A -85,B 0,C 180,E1 -29438.73,E2 -29438.73} C_VEL
LIN {X 0,Y 49.914,Z 553.404,A -85,B 0,C 180,E1 -29454.986,E2 -29454.986} C_VEL
LIN {X 0,Y 52.772,Z 552.108,A -85,B 0,C 180,E1 -29462.188,E2 -29462.188} C_VEL
LIN {X 0,Y 58.815,Z 549.252,A -85,B 0,C 180,E1 -29471.086,E2 -29471.086} C_VEL
LIN {X 0,Y 65.775,Z 545.412,A -85,B 0,C 180,E1 -29478.412,E2 -29478.412} C_VEL
LIN {X 0,Y 73.602,Z 540.316,A -85,B 0,C 180,E1 -29484.723,E2 -29484.723} C_VEL
LIN {X 0,Y 83.024,Z 533.058,A -85,B 0,C 180,E1 -29490.187,E2 -29490.187} C_VEL
LIN {X 0,Y 91.723,Z 525.016,A -85,B 0,C 180,E1 -29494.196,E2 -29494.196} C_VEL
LIN {X 0,Y 99.161,Z 516.778,A -85,B 0,C 180,E1 -29497.125,E2 -29497.125} C_VEL
LIN {X 0,Y 106.014,Z 507.718,A -85,B 0,C 180,E1 -29499.451,E2 -29499.451} C_VEL
LIN {X 0,Y 113.27,Z 496.123,A -85,B 0,C 180,E1 -29501.363,E2 -29501.363} C_VEL
LIN {X 0,Y 118.827,Z 484.781,A -85,B 0,C 180,E1 -29502.881,E2 -29502.881} C_VEL
LIN {X 0,Y 123.227,Z 473.062,A -85,B 0,C 180,E1 -29503.983,E2 -29503.983} C_VEL
LIN {X 0,Y 126.631,Z 459.865,A -85,B 0,C 180,E1 -29505.066,E2 -29505.066} C_VEL
LIN {X 0,Y 127.327,Z 456.081,A -85,B 0,C 180,E1 -29505.358,E2 -29505.358} C_VEL
LIN {X 0,Y 126.559,Z 452.89,A -85,B 0,C 180,E1 -29508.387,E2 -29508.387} C_VEL
LIN {X 0,Y 125.651,Z 449.536,A -85,B 0,C 180,E1 -29512.77,E2 -29512.77} C_VEL
LIN {X 0,Y 125.196,Z 447.244,A -85,B 0,C 180,E1 -29518.391,E2 -29518.391} C_VEL
LIN {X 0,Y 125.206,Z 447.823,A -85,B 0,C 180,E1 -29521.206,E2 -29521.206} C_VEL
LIN {X 0,Y 125.65,Z 449.608,A -85,B 0,C 180,E1 -29525.315,E2 -29525.315} C_VEL
LIN {X 0,Y 126.132,Z 454.396,A -85,B 0,C 180,E1 -29528.814,E2 -29528.814} C_VEL
LIN {X 0,Y 126.528,Z 458.902,A -85,B 0,C 180,E1 -29531.261,E2 -29531.261} C_VEL
LIN {X 0,Y 124.386,Z 472.011,A -85,B 0,C 180,E1 -29532.595,E2 -29532.595} C_VEL
LIN {X 0,Y 120.436,Z 484.857,A -85,B 0,C 180,E1 -29533.277,E2 -29533.277} C_VEL
LIN {X 0,Y 115.293,Z 497.023,A -85,B 0,C 180,E1 -29534.113,E2 -29534.113} C_VEL
LIN {X 0,Y 109.297,Z 508.224,A -85,B 0,C 180,E1 -29535.31,E2 -29535.31} C_VEL
LIN {X 0,Y 101.851,Z 519.145,A -85,B 0,C 180,E1 -29536.785,E2 -29536.785} C_VEL
LIN {X 0,Y 94.582,Z 528.114,A -85,B 0,C 180,E1 -29538.668,E2 -29538.668} C_VEL
LIN {X 0,Y 85.017,Z 537.865,A -85,B 0,C 180,E1 -29541.57,E2 -29541.57} C_VEL
LIN {X 0,Y 75.844,Z 545.687,A -85,B 0,C 180,E1 -29545.384,E2 -29545.384} C_VEL
LIN {X 0,Y 65.767,Z 552.961,A -85,B 0,C 180,E1 -29551.253,E2 -29551.253} C_VEL
LIN {X 0,Y 58.009,Z 557.873,A -85,B 0,C 180,E1 -29558.049,E2 -29558.049} C_VEL
LIN {X 0,Y 51.341,Z 561.683,A -85,B 0,C 180,E1 -29566.809,E2 -29566.809} C_VEL
LIN {X 0,Y 47.776,Z 563.691,A -85,B 0,C 180,E1 -29573.956,E2 -29573.956} C_VEL
LIN {X 0,Y 43.608,Z 566.422,A -85,B 0,C 180,E1 -29591.197,E2 -29591.197} C_VEL
LIN {X 0,Y 43.859,Z 567.583,A -85,B 0,C 180,E1 -29610,E2 -29610} C_VEL
LIN {X 0,Y 43.601,Z 566.388,A -85,B 0,C 180,E1 -29628.806,E2 -29628.806} C_VEL
LIN {X 0,Y 47.769,Z 563.624,A -85,B 0,C 180,E1 -29646.05,E2 -29646.05} C_VEL
LIN {X 0,Y 53.392,Z 560.443,A -85,B 0,C 180,E1 -29656.382,E2 -29656.382} C_VEL
LIN {X 0,Y 60.586,Z 556.171,A -85,B 0,C 180,E1 -29664.55,E2 -29664.55} C_VEL
LIN {X 0,Y 69.959,Z 549.878,A -85,B 0,C 180,E1 -29671.522,E2 -29671.522} C_VEL
LIN {X 0,Y 78.85,Z 543.027,A -85,B 0,C 180,E1 -29676.005,E2 -29676.005} C_VEL
LIN {X 0,Y 88.167,Z 534.584,A -85,B 0,C 180,E1 -29679.488,E2 -29679.488} C_VEL
LIN {X 0,Y 96.215,Z 525.975,A -85,B 0,C 180,E1 -29681.725,E2 -29681.725} C_VEL
LIN {X 0,Y 103.513,Z 516.523,A -85,B 0,C 180,E1 -29683.535,E2 -29683.535} C_VEL
LIN {X 0,Y 110.61,Z 505.403,A -85,B 0,C 180,E1 -29684.984,E2 -29684.984} C_VEL
LIN {X 0,Y 116.494,Z 493.872,A -85,B 0,C 180,E1 -29686.055,E2 -29686.055} C_VEL
LIN {X 0,Y 121.145,Z 482.017,A -85,B 0,C 180,E1 -29686.843,E2 -29686.843} C_VEL
LIN {X 0,Y 124.357,Z 470.618,A -85,B 0,C 180,E1 -29687.51,E2 -29687.51} C_VEL
LIN {X 0,Y 126.241,Z 458.523,A -85,B 0,C 180,E1 -29688.763,E2 -29688.763} C_VEL
LIN {X 0,Y 125.725,Z 452.761,A -85,B 0,C 180,E1 -29691.967,E2 -29691.967} C_VEL
LIN {X 0,Y 125.338,Z 449.236,A -85,B 0,C 180,E1 -29694.772,E2 -29694.772} C_VEL
LIN {X 0,Y 124.903,Z 446.904,A -85,B 0,C 180,E1 -29700,E2 -29700} C_VEL
LIN {X 0,Y 124.898,Z 446.949,A -85,B 0,C 180,E1 -29702.016,E2 -29702.016} C_VEL
LIN {X 0,Y 125.498,Z 449.885,A -85,B 0,C 180,E1 -29708.251,E2 -29708.251} C_VEL
LIN {X 0,Y 126.401,Z 453.159,A -85,B 0,C 180,E1 -29712.238,E2 -29712.238} C_VEL
LIN {X 0,Y 127.056,Z 455.843,A -85,B 0,C 180,E1 -29714.761,E2 -29714.761} C_VEL
LIN {X 0,Y 124.479,Z 467.518,A -85,B 0,C 180,E1 -29715.567,E2 -29715.567} C_VEL
LIN {X 0,Y 120.74,Z 479.244,A -85,B 0,C 180,E1 -29716.651,E2 -29716.651} C_VEL
LIN {X 0,Y 115.609,Z 491.037,A -85,B 0,C 180,E1 -29718.031,E2 -29718.031} C_VEL
LIN {X 0,Y 109.971,Z 501.193,A -85,B 0,C 180,E1 -29719.504,E2 -29719.504} C_VEL
LIN {X 0,Y 106.527,Z 506.52,A -85,B 0,C 180,E1 -29720.484,E2 -29720.484} C_VEL
LIN {X 0,Y 101.733,Z 512.724,A -85,B 0,C 180,E1 -29721.096,E2 -29721.096} C_VEL
LIN {X 0,Y 96.376,Z 518.598,A -85,B 0,C 180,E1 -29721.319,E2 -29721.319} C_VEL
LIN {X 0,Y 89.318,Z 525.414,A -85,B 0,C 180,E1 -29721.965,E2 -29721.965} C_VEL
LIN {X 0,Y 85.139,Z 529.183,A -85,B 0,C 180,E1 -29723.105,E2 -29723.105} C_VEL
LIN {X 0,Y 76.628,Z 536.241,A -85,B 0,C 180,E1 -29726.885,E2 -29726.885} C_VEL
LIN {X 0,Y 66.746,Z 543.034,A -85,B 0,C 180,E1 -29732.612,E2 -29732.612} C_VEL
LIN {X 0,Y 58.687,Z 547.635,A -85,B 0,C 180,E1 -29738.887,E2 -29738.887} C_VEL
LIN {X 0,Y 51.258,Z 551.183,A -85,B 0,C 180,E1 -29746.722,E2 -29746.722} C_VEL
LIN {X 0,Y 46.988,Z 553.003,A -85,B 0,C 180,E1 -29753.254,E2 -29753.254} C_VEL
LIN {X 0,Y 43.652,Z 554.325,A -85,B 0,C 180,E1 -29761.119,E2 -29761.119} C_VEL
LIN {X 0,Y 39.371,Z 555.863,A -85,B 0,C 180,E1 -29779.717,E2 -29779.717} C_VEL
LIN {X 0,Y 38.801,Z 556.081,A -85,B 0,C 180,E1 -29790,E2 -29790} C_VEL
LIN {X 0,Y 39.37,Z 555.887,A -85,B 0,C 180,E1 -29800.283,E2 -29800.283} C_VEL
LIN {X 0,Y 43.643,Z 554.382,A -85,B 0,C 180,E1 -29818.888,E2 -29818.888} C_VEL
LIN {X 0,Y 46.971,Z 553.086,A -85,B 0,C 180,E1 -29826.762,E2 -29826.762} C_VEL
LIN {X 0,Y 53.717,Z 550.229,A -85,B 0,C 180,E1 -29836.019,E2 -29836.019} C_VEL
LIN {X 0,Y 61.335,Z 546.389,A -85,B 0,C 180,E1 -29843.328,E2 -29843.328} C_VEL
LIN {X 0,Y 69.779,Z 541.293,A -85,B 0,C 180,E1 -29849.439,E2 -29849.439} C_VEL
LIN {X 0,Y 79.763,Z 534.034,A -85,B 0,C 180,E1 -29854.571,E2 -29854.571} C_VEL
LIN {X 0,Y 88.889,Z 525.992,A -85,B 0,C 180,E1 -29858.279,E2 -29858.279} C_VEL
LIN {X 0,Y 96.645,Z 517.753,A -85,B 0,C 180,E1 -29860.968,E2 -29860.968} C_VEL
LIN {X 0,Y 103.756,Z 508.693,A -85,B 0,C 180,E1 -29863.088,E2 -29863.088} C_VEL
LIN {X 0,Y 111.222,Z 497.098,A -85,B 0,C 180,E1 -29864.797,E2 -29864.797} C_VEL
LIN {X 0,Y 116.866,Z 485.937,A -85,B 0,C 180,E1 -29866.153,E2 -29866.153} C_VEL
LIN {X 0,Y 121.476,Z 474.031,A -85,B 0,C 180,E1 -29867.171,E2 -29867.171} C_VEL
LIN {X 0,Y 124.989,Z 460.9,A -85,B 0,C 180,E1 -29868.175,E2 -29868.175} C_VEL
LIN {X 0,Y 125.053,Z 460.432,A -85,B 0,C 180,E1 -29868.307,E2 -29868.307} C_VEL
LIN {X 0,Y 124.463,Z 456.737,A -85,B 0,C 180,E1 -29872.904,E2 -29872.904} C_VEL
LIN {X 0,Y 124.233,Z 454.425,A -85,B 0,C 180,E1 -29878.379,E2 -29878.379} C_VEL
LIN {X 0,Y 124.258,Z 454.943,A -85,B 0,C 180,E1 -29881.215,E2 -29881.215} C_VEL
LIN {X 0,Y 124.516,Z 456.368,A -85,B 0,C 180,E1 -29884.35,E2 -29884.35} C_VEL
LIN {X 0,Y 124.619,Z 461.019,A -85,B 0,C 180,E1 -29887.595,E2 -29887.595} C_VEL
LIN {X 0,Y 124.626,Z 462.407,A -85,B 0,C 180,E1 -29888.36,E2 -29888.36} C_VEL
LIN {X 0,Y 122.454,Z 473.138,A -85,B 0,C 180,E1 -29889.455,E2 -29889.455} C_VEL
LIN {X 0,Y 118.6,Z 484.949,A -85,B 0,C 180,E1 -29889.993,E2 -29889.993} C_VEL
LIN {X 0,Y 113.592,Z 496.404,A -85,B 0,C 180,E1 -29890.657,E2 -29890.657} C_VEL
LIN {X 0,Y 107.639,Z 507.24,A -85,B 0,C 180,E1 -29891.659,E2 -29891.659} C_VEL
LIN {X 0,Y 100.032,Z 518.161,A -85,B 0,C 180,E1 -29892.889,E2 -29892.889} C_VEL
LIN {X 0,Y 92.555,Z 527.13,A -85,B 0,C 180,E1 -29894.505,E2 -29894.505} C_VEL
LIN {X 0,Y 82.657,Z 536.873,A -85,B 0,C 180,E1 -29896.957,E2 -29896.957} C_VEL
LIN {X 0,Y 73.069,Z 544.695,A -85,B 0,C 180,E1 -29900.319,E2 -29900.319} C_VEL
LIN {X 0,Y 62.359,Z 551.968,A -85,B 0,C 180,E1 -29905.631,E2 -29905.631} C_VEL
LIN {X 0,Y 54.956,Z 556.288,A -85,B 0,C 180,E1 -29911.086,E2 -29911.086} C_VEL
LIN {X 0,Y 46.37,Z 560.685,A -85,B 0,C 180,E1 -29920.729,E2 -29920.729} C_VEL
LIN {X 0,Y 42.185,Z 562.693,A -85,B 0,C 180,E1 -29928.212,E2 -29928.212} C_VEL
LIN {X 0,Y 36.899,Z 565.425,A -85,B 0,C 180,E1 -29947.609,E2 -29947.609} C_VEL
LIN {X 0,Y 36.135,Z 566.208,A -85,B 0,C 180,E1 -29958.785,E2 -29958.785} C_VEL
LIN {X 0,Y 36.716,Z 566.589,A -85,B 0,C 180,E1 -29970,E2 -29970} C_VEL
LIN {X 0,Y 36.89,Z 565.391,A -85,B 0,C 180,E1 -29992.396,E2 -29992.396} C_VEL
LIN {X 0,Y 42.181,Z 562.625,A -85,B 0,C 180,E1 -30011.794,E2 -30011.794} C_VEL
LIN {X 0,Y 48.737,Z 559.448,A -85,B 0,C 180,E1 -30022.476,E2 -30022.476} C_VEL
LIN {X 0,Y 56.617,Z 555.247,A -85,B 0,C 180,E1 -30030.332,E2 -30030.332} C_VEL
LIN {X 0,Y 66.843,Z 548.881,A -85,B 0,C 180,E1 -30036.922,E2 -30036.922} C_VEL
LIN {X 0,Y 76.221,Z 542.029,A -85,B 0,C 180,E1 -30040.925,E2 -30040.925} C_VEL
LIN {X 0,Y 85.939,Z 533.595,A -85,B 0,C 180,E1 -30043.922,E2 -30043.922} C_VEL
LIN {X 0,Y 94.224,Z 524.98,A -85,B 0,C 180,E1 -30045.843,E2 -30045.843} C_VEL
LIN {X 0,Y 101.73,Z 515.532,A -85,B 0,C 180,E1 -30047.37,E2 -30047.37} C_VEL
LIN {X 0,Y 108.687,Z 504.904,A -85,B 0,C 180,E1 -30048.562,E2 -30048.562} C_VEL
LIN {X 0,Y 115.055,Z 492.722,A -85,B 0,C 180,E1 -30049.519,E2 -30049.519} C_VEL
LIN {X 0,Y 120.081,Z 479.917,A -85,B 0,C 180,E1 -30050.217,E2 -30050.217} C_VEL
LIN {X 0,Y 122.542,Z 471.49,A -85,B 0,C 180,E1 -30050.683,E2 -30050.683} C_VEL
LIN {X 0,Y 124.345,Z 462.028,A -85,B 0,C 180,E1 -30051.694,E2 -30051.694} C_VEL
LIN {X 0,Y 124.278,Z 457.821,A -85,B 0,C 180,E1 -30054.321,E2 -30054.321} C_VEL
LIN {X 0,Y 124.205,Z 455.773,A -85,B 0,C 180,E1 -30055.944,E2 -30055.944} C_VEL
LIN {X 0,Y 123.961,Z 454.071,A -85,B 0,C 180,E1 -30060,E2 -30060} C_VEL
LIN {X 0,Y 123.936,Z 454.149,A -85,B 0,C 180,E1 -30062.031,E2 -30062.031} C_VEL
LIN {X 0,Y 124.184,Z 456.573,A -85,B 0,C 180,E1 -30067.316,E2 -30067.316} C_VEL
LIN {X 0,Y 124.705,Z 459.775,A -85,B 0,C 180,E1 -30071.315,E2 -30071.315} C_VEL
